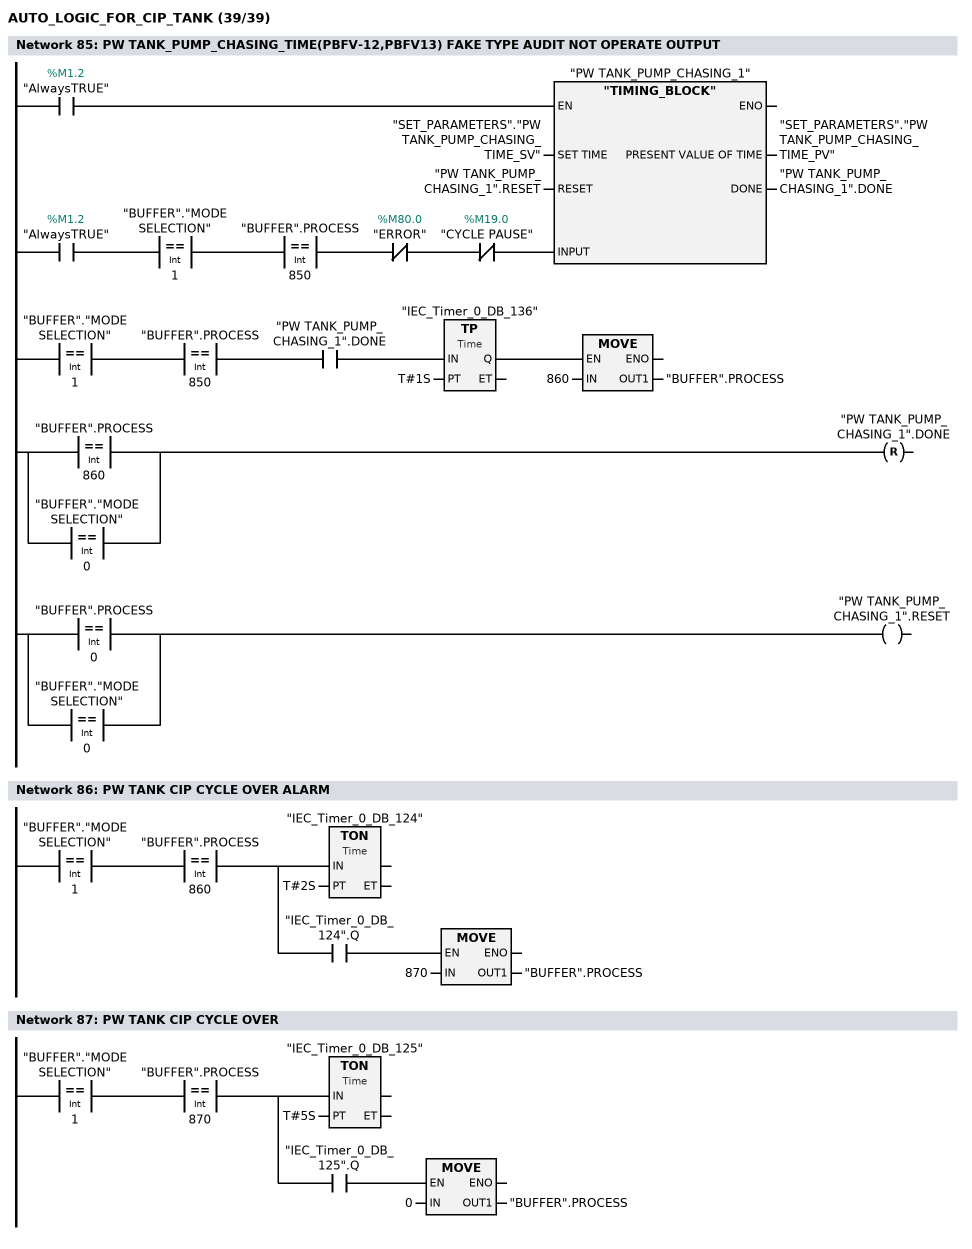
   RUNG wire#powerrail
      Contact( "AlwaysTRUE" )
      "PW TANK_PUMP_CHASING_1"(INPUT := wire#w1, "SET TIME" := "SET_PARAMETERS"."PW TANK_PUMP_CHASING_TIME_SV", RESET := "PW TANK_PUMP_CHASING_1".RESET, "PRESENT VALUE OF TIME" => "SET_PARAMETERS"."PW TANK_PUMP_CHASING_TIME_PV", DONE => "PW TANK_PUMP_CHASING_1".DONE)
   END_RUNG
   RUNG wire#powerrail
      Contact( "AlwaysTRUE" )
      { S7_Templates := "SrcType := Int" } EQ_Contact(in1 := "BUFFER"."MODE SELECTION", in2 := 1)
      { S7_Templates := "SrcType := Int" } EQ_Contact(in1 := "BUFFER".PROCESS, in2 := 850)
      I_Contact( "ERROR" )
      I_Contact( "CYCLE PAUSE" )
   END_RUNG wire#w1
   RUNG wire#powerrail
      { S7_Templates := "SrcType := Int" } EQ_Contact(in1 := "BUFFER"."MODE SELECTION", in2 := 1)
      { S7_Templates := "SrcType := Int" } EQ_Contact(in1 := "BUFFER".PROCESS, in2 := 850)
      Contact( "PW TANK_PUMP_CHASING_1".DONE )
      { S7_Templates := "time_type := Time" } "IEC_Timer_0_DB_136".TP(pt := T#1S, et =>)
      Move(in := 860, out1 => "BUFFER".PROCESS)
   END_RUNG
   RUNG wire#powerrail
      { S7_Templates := "SrcType := Int" } EQ_Contact(in1 := "BUFFER".PROCESS, in2 := 860)
      wire#w2
      R_Coil( "PW TANK_PUMP_CHASING_1".DONE )
   END_RUNG
   RUNG wire#powerrail
      { S7_Templates := "SrcType := Int" } EQ_Contact(in1 := "BUFFER"."MODE SELECTION", in2 := 0)
   END_RUNG wire#w2
   RUNG wire#powerrail
      { S7_Templates := "SrcType := Int" } EQ_Contact(in1 := "BUFFER".PROCESS, in2 := 0)
      wire#w3
      Coil( "PW TANK_PUMP_CHASING_1".RESET )
   END_RUNG
   RUNG wire#powerrail
      { S7_Templates := "SrcType := Int" } EQ_Contact(in1 := "BUFFER"."MODE SELECTION", in2 := 0)
   END_RUNG wire#w3
   // the same network as SCL:
   IF "AlwaysTRUE" THEN
       "PW TANK_PUMP_CHASING_1"("SET TIME" := "SET_PARAMETERS"."PW TANK_PUMP_CHASING_TIME_SV",   // "TIMING_BLOCK"
                               RESET := "PW TANK_PUMP_CHASING_1".RESET,
                               INPUT := "AlwaysTRUE" AND ("BUFFER"."MODE SELECTION" = 1) AND ("BUFFER".PROCESS = 850) AND NOT "ERROR" AND NOT "CYCLE PAUSE",
                               "PRESENT VALUE OF TIME" => "SET_PARAMETERS"."PW TANK_PUMP_CHASING_TIME_PV",
                               DONE => "PW TANK_PUMP_CHASING_1".DONE);
   END_IF;
   "IEC_Timer_0_DB_136".TP(IN := ("BUFFER"."MODE SELECTION" = 1) AND ("BUFFER".PROCESS = 850) AND "PW TANK_PUMP_CHASING_1".DONE,
                           PT := T#1S);
   IF "IEC_Timer_0_DB_136".Q THEN "BUFFER".PROCESS := 860; END_IF;
   IF ("BUFFER".PROCESS = 860) OR ("BUFFER"."MODE SELECTION" = 0) THEN
       "PW TANK_PUMP_CHASING_1".DONE := FALSE;
   END_IF;
   "PW TANK_PUMP_CHASING_1".RESET := ("BUFFER".PROCESS = 0) OR ("BUFFER"."MODE SELECTION" = 0);
END_REGION

REGION Network 86: PW TANK CIP CYCLE OVER ALARM
   RUNG wire#powerrail
      { S7_Templates := "SrcType := Int" } EQ_Contact(in1 := "BUFFER"."MODE SELECTION", in2 := 1)
      { S7_Templates := "SrcType := Int" } EQ_Contact(in1 := "BUFFER".PROCESS, in2 := 860)
      wire#w1
      { S7_Templates := "time_type := Time" } "IEC_Timer_0_DB_124".TON(pt := T#2S, et =>)
   END_RUNG
   RUNG wire#w1
      Contact( "IEC_Timer_0_DB_124".Q )
      Move(in := 870, out1 => "BUFFER".PROCESS)
   END_RUNG
   // the same network as SCL:
   #_w1 := ("BUFFER"."MODE SELECTION" = 1) AND ("BUFFER".PROCESS = 860);
   "IEC_Timer_0_DB_124".TON(IN := #_w1, PT := T#2S);
   IF #_w1 AND "IEC_Timer_0_DB_124".Q THEN "BUFFER".PROCESS := 870; END_IF;
END_REGION

REGION Network 87: PW TANK CIP CYCLE OVER
   RUNG wire#powerrail
      { S7_Templates := "SrcType := Int" } EQ_Contact(in1 := "BUFFER"."MODE SELECTION", in2 := 1)
      { S7_Templates := "SrcType := Int" } EQ_Contact(in1 := "BUFFER".PROCESS, in2 := 870)
      wire#w1
      { S7_Templates := "time_type := Time" } "IEC_Timer_0_DB_125".TON(pt := T#5S, et =>)
   END_RUNG
   RUNG wire#w1
      Contact( "IEC_Timer_0_DB_125".Q )
      Move(in := 0, out1 => "BUFFER".PROCESS)
   END_RUNG
   // the same network as SCL:
   #_w1 := ("BUFFER"."MODE SELECTION" = 1) AND ("BUFFER".PROCESS = 870);
   "IEC_Timer_0_DB_125".TON(IN := #_w1, PT := T#5S);
   IF #_w1 AND "IEC_Timer_0_DB_125".Q THEN "BUFFER".PROCESS := 0; END_IF;
END_REGION
END_FUNCTION

FUNCTION_BLOCK "TIMING_BLOCK"   // FB2, LAD
{ S7_Optimized_Access := 'TRUE' }
// stored: MemoryReserve 100, SetENOAutomatically false
   VAR_INPUT
      "SET TIME" : Int;
      RESET : Bool;
      INPUT : Bool;
   END_VAR
   VAR_OUTPUT
      "PRESENT VALUE OF TIME" : Int;
      DONE : Bool;
   END_VAR
   VAR
      "TIMER 1" { S7_SetPoint := 'True'} : IEC_TIMER;
   END_VAR
   VAR RETAIN
      "COUNTER1 1" { S7_SetPoint := 'True'} : IEC_COUNTER;
   END_VAR
   VAR_TEMP   // added for the SCL form of the ladder/FBD networks
      _w1 : Bool;
      _w2 : Bool;
   END_VAR
BEGIN

REGION Network 1
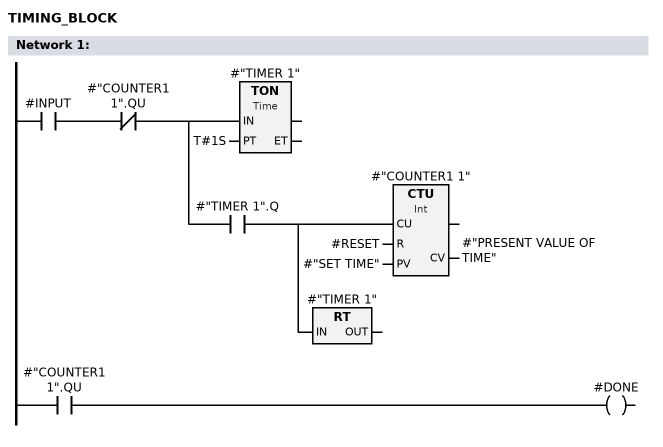
   RUNG wire#powerrail
      Contact( #INPUT )
      I_Contact( #"COUNTER1 1".QU )
      wire#w1
      { S7_Templates := "time_type := Time" } #"TIMER 1".TON(pt := T#1S, et =>)
   END_RUNG
   RUNG wire#w1
      Contact( #"TIMER 1".Q )
      wire#w2
      { S7_Templates := "value_type := Int" } #"COUNTER1 1".CTU(r := #RESET, pv := #"SET TIME", cv => #"PRESENT VALUE OF TIME")
   END_RUNG
   RUNG wire#w2
      RT_Coil( #"TIMER 1" )
   END_RUNG
   RUNG wire#powerrail
      Contact( #"COUNTER1 1".QU )
      Coil( #DONE )
   END_RUNG
   // the same network as SCL:
   #_w1 := #INPUT AND NOT #"COUNTER1 1".QU;
   #"TIMER 1".TON(IN := #_w1, PT := T#1S);
   #_w2 := #_w1 AND #"TIMER 1".Q;
   #"COUNTER1 1".CTU(CU := #_w2, R := #RESET, PV := #"SET TIME", CV => #"PRESENT VALUE OF TIME");
   IF #_w2 THEN RESET_TIMER(#"TIMER 1"); END_IF;
   #DONE := #"COUNTER1 1".QU;
END_REGION
END_FUNCTION_BLOCK

FUNCTION "POPUP" : Void   // FC6, LAD
{ S7_Optimized_Access := 'TRUE' }
// stored: SetENOAutomatically false
   VAR_TEMP   // added for the SCL form of the ladder/FBD networks
      _w1 : Bool;
      _w2 : Bool;
   END_VAR
BEGIN

REGION Network 1: RINSE-1_START
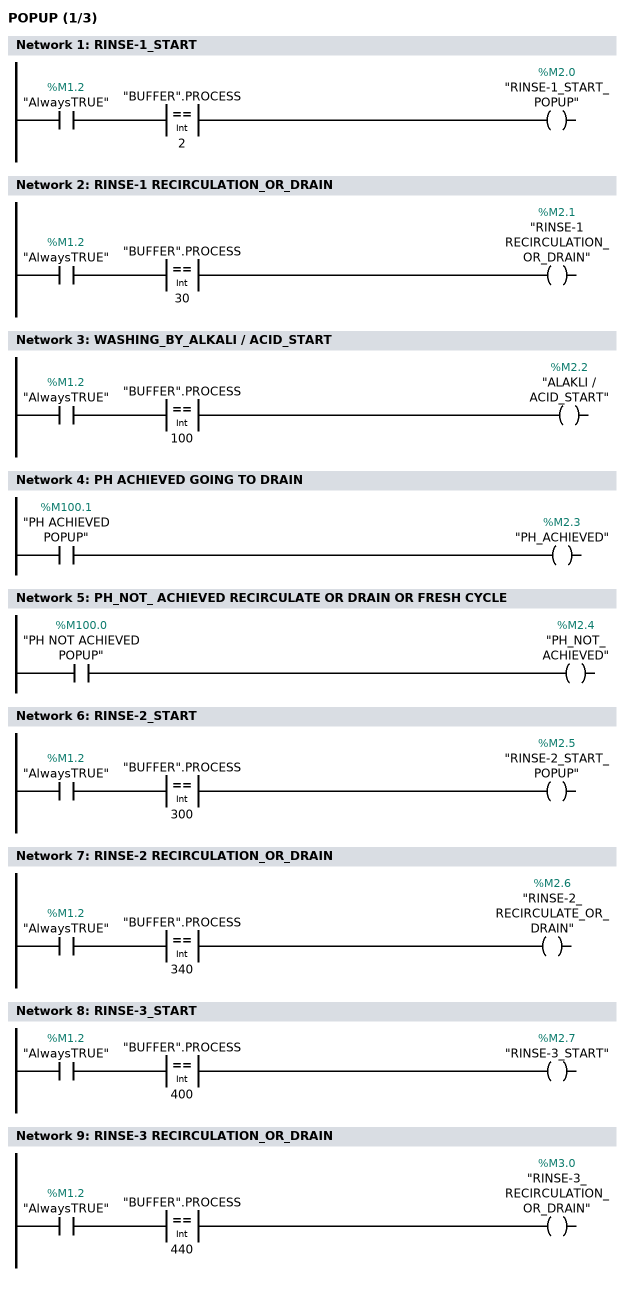
   RUNG wire#powerrail
      Contact( "AlwaysTRUE" )
      { S7_Templates := "SrcType := Int" } EQ_Contact(in1 := "BUFFER".PROCESS, in2 := 2)
      Coil( "RINSE-1_START_POPUP" )
   END_RUNG
   // the same network as SCL:
   "RINSE-1_START_POPUP" := "AlwaysTRUE" AND ("BUFFER".PROCESS = 2);
END_REGION

REGION Network 2: RINSE-1 RECIRCULATION_OR_DRAIN
   RUNG wire#powerrail
      Contact( "AlwaysTRUE" )
      { S7_Templates := "SrcType := Int" } EQ_Contact(in1 := "BUFFER".PROCESS, in2 := 30)
      Coil( "RINSE-1 RECIRCULATION_OR_DRAIN" )
   END_RUNG
   // the same network as SCL:
   "RINSE-1 RECIRCULATION_OR_DRAIN" := "AlwaysTRUE" AND ("BUFFER".PROCESS = 30);
END_REGION

REGION Network 3: WASHING_BY_ALKALI / ACID_START
   RUNG wire#powerrail
      Contact( "AlwaysTRUE" )
      { S7_Templates := "SrcType := Int" } EQ_Contact(in1 := "BUFFER".PROCESS, in2 := 100)
      Coil( "ALAKLI / ACID_START" )
   END_RUNG
   // the same network as SCL:
   "ALAKLI / ACID_START" := "AlwaysTRUE" AND ("BUFFER".PROCESS = 100);
END_REGION

REGION Network 4: PH ACHIEVED GOING TO DRAIN
   RUNG wire#powerrail
      Contact( "PH ACHIEVED POPUP" )
      Coil( "PH_ACHIEVED" )
   END_RUNG
   // the same network as SCL:
   "PH_ACHIEVED" := "PH ACHIEVED POPUP";
END_REGION

REGION Network 5: PH_NOT_ ACHIEVED RECIRCULATE OR DRAIN OR FRESH CYCLE
   RUNG wire#powerrail
      Contact( "PH NOT ACHIEVED POPUP" )
      Coil( "PH_NOT_ACHIEVED" )
   END_RUNG
   // the same network as SCL:
   "PH_NOT_ACHIEVED" := "PH NOT ACHIEVED POPUP";
END_REGION

REGION Network 6: RINSE-2_START
   RUNG wire#powerrail
      Contact( "AlwaysTRUE" )
      { S7_Templates := "SrcType := Int" } EQ_Contact(in1 := "BUFFER".PROCESS, in2 := 300)
      Coil( "RINSE-2_START_POPUP" )
   END_RUNG
   // the same network as SCL:
   "RINSE-2_START_POPUP" := "AlwaysTRUE" AND ("BUFFER".PROCESS = 300);
END_REGION

REGION Network 7: RINSE-2 RECIRCULATION_OR_DRAIN
   RUNG wire#powerrail
      Contact( "AlwaysTRUE" )
      { S7_Templates := "SrcType := Int" } EQ_Contact(in1 := "BUFFER".PROCESS, in2 := 340)
      Coil( "RINSE-2_RECIRCULATE_OR_DRAIN" )
   END_RUNG
   // the same network as SCL:
   "RINSE-2_RECIRCULATE_OR_DRAIN" := "AlwaysTRUE" AND ("BUFFER".PROCESS = 340);
END_REGION

REGION Network 8: RINSE-3_START
   RUNG wire#powerrail
      Contact( "AlwaysTRUE" )
      { S7_Templates := "SrcType := Int" } EQ_Contact(in1 := "BUFFER".PROCESS, in2 := 400)
      Coil( "RINSE-3_START" )
   END_RUNG
   // the same network as SCL:
   "RINSE-3_START" := "AlwaysTRUE" AND ("BUFFER".PROCESS = 400);
END_REGION

REGION Network 9: RINSE-3 RECIRCULATION_OR_DRAIN
   RUNG wire#powerrail
      Contact( "AlwaysTRUE" )
      { S7_Templates := "SrcType := Int" } EQ_Contact(in1 := "BUFFER".PROCESS, in2 := 440)
      Coil( "RINSE-3_RECIRCULATION_OR_DRAIN" )
   END_RUNG
   // the same network as SCL:
   "RINSE-3_RECIRCULATION_OR_DRAIN" := "AlwaysTRUE" AND ("BUFFER".PROCESS = 440);
END_REGION

REGION Network 10: FINAL_RINSE_START
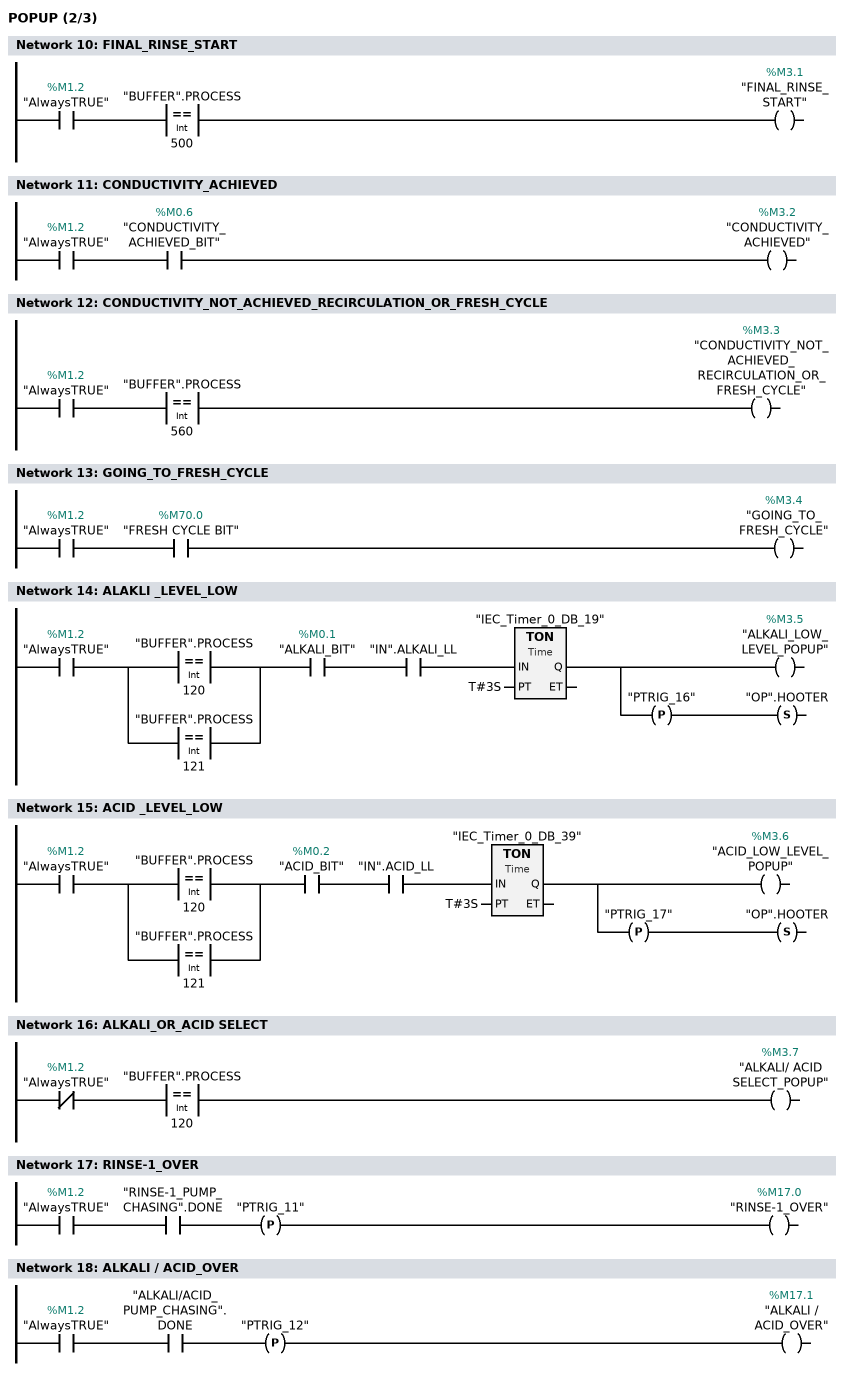
   RUNG wire#powerrail
      Contact( "AlwaysTRUE" )
      { S7_Templates := "SrcType := Int" } EQ_Contact(in1 := "BUFFER".PROCESS, in2 := 500)
      Coil( "FINAL_RINSE_START" )
   END_RUNG
   // the same network as SCL:
   "FINAL_RINSE_START" := "AlwaysTRUE" AND ("BUFFER".PROCESS = 500);
END_REGION

REGION Network 11: CONDUCTIVITY_ACHIEVED
   RUNG wire#powerrail
      Contact( "AlwaysTRUE" )
      Contact( "CONDUCTIVITY_ACHIEVED_BIT" )
      Coil( "CONDUCTIVITY_ACHIEVED" )
   END_RUNG
   // the same network as SCL:
   "CONDUCTIVITY_ACHIEVED" := "AlwaysTRUE" AND "CONDUCTIVITY_ACHIEVED_BIT";
END_REGION

REGION Network 12: CONDUCTIVITY_NOT_ACHIEVED_RECIRCULATION_OR_FRESH_CYCLE
   RUNG wire#powerrail
      Contact( "AlwaysTRUE" )
      { S7_Templates := "SrcType := Int" } EQ_Contact(in1 := "BUFFER".PROCESS, in2 := 560)
      Coil( "CONDUCTIVITY_NOT_ACHIEVED_RECIRCULATION_OR_FRESH_CYCLE" )
   END_RUNG
   // the same network as SCL:
   "CONDUCTIVITY_NOT_ACHIEVED_RECIRCULATION_OR_FRESH_CYCLE" := "AlwaysTRUE" AND ("BUFFER".PROCESS = 560);
END_REGION

REGION Network 13: GOING_TO_FRESH_CYCLE
   RUNG wire#powerrail
      Contact( "AlwaysTRUE" )
      Contact( "FRESH CYCLE BIT" )
      Coil( "GOING_TO_FRESH_CYCLE" )
   END_RUNG
   // the same network as SCL:
   "GOING_TO_FRESH_CYCLE" := "AlwaysTRUE" AND "FRESH CYCLE BIT";
END_REGION

REGION Network 14: ALAKLI _LEVEL_LOW
   RUNG wire#powerrail
      Contact( "AlwaysTRUE" )
      wire#w1
      { S7_Templates := "SrcType := Int" } EQ_Contact(in1 := "BUFFER".PROCESS, in2 := 120)
      wire#w2
      Contact( "ALKALI_BIT" )
      Contact( "IN".ALKALI_LL )
      { S7_Templates := "time_type := Time" } "IEC_Timer_0_DB_19".TON(pt := T#3S, et =>)
      wire#w3
      Coil( "ALKALI_LOW_LEVEL_POPUP" )
   END_RUNG
   RUNG wire#w1
      { S7_Templates := "SrcType := Int" } EQ_Contact(in1 := "BUFFER".PROCESS, in2 := 121)
   END_RUNG wire#w2
   RUNG wire#w3
      P_Trig( "PTRIG_16" )
      S_Coil( "OP".HOOTER )
   END_RUNG
   // the same network as SCL:
   "IEC_Timer_0_DB_19".TON(IN := "AlwaysTRUE" AND (("BUFFER".PROCESS = 120) OR ("BUFFER".PROCESS = 121)) AND "ALKALI_BIT" AND "IN".ALKALI_LL,
                           PT := T#3S);
   "ALKALI_LOW_LEVEL_POPUP" := "IEC_Timer_0_DB_19".Q;
   #_w1 := "IEC_Timer_0_DB_19".Q AND NOT "PTRIG_16";   // rising edge
   "PTRIG_16" := "IEC_Timer_0_DB_19".Q;
   IF #_w1 THEN "OP".HOOTER := TRUE; END_IF;
END_REGION

REGION Network 15: ACID _LEVEL_LOW
   RUNG wire#powerrail
      Contact( "AlwaysTRUE" )
      wire#w1
      { S7_Templates := "SrcType := Int" } EQ_Contact(in1 := "BUFFER".PROCESS, in2 := 120)
      wire#w2
      Contact( "ACID_BIT" )
      Contact( "IN".ACID_LL )
      { S7_Templates := "time_type := Time" } "IEC_Timer_0_DB_39".TON(pt := T#3S, et =>)
      wire#w3
      Coil( "ACID_LOW_LEVEL_POPUP" )
   END_RUNG
   RUNG wire#w1
      { S7_Templates := "SrcType := Int" } EQ_Contact(in1 := "BUFFER".PROCESS, in2 := 121)
   END_RUNG wire#w2
   RUNG wire#w3
      P_Trig( "PTRIG_17" )
      S_Coil( "OP".HOOTER )
   END_RUNG
   // the same network as SCL:
   "IEC_Timer_0_DB_39".TON(IN := "AlwaysTRUE" AND (("BUFFER".PROCESS = 120) OR ("BUFFER".PROCESS = 121)) AND "ACID_BIT" AND "IN".ACID_LL,
                           PT := T#3S);
   "ACID_LOW_LEVEL_POPUP" := "IEC_Timer_0_DB_39".Q;
   #_w1 := "IEC_Timer_0_DB_39".Q AND NOT "PTRIG_17";   // rising edge
   "PTRIG_17" := "IEC_Timer_0_DB_39".Q;
   IF #_w1 THEN "OP".HOOTER := TRUE; END_IF;
END_REGION

REGION Network 16: ALKALI_OR_ACID SELECT
   RUNG wire#powerrail
      I_Contact( "AlwaysTRUE" )
      { S7_Templates := "SrcType := Int" } EQ_Contact(in1 := "BUFFER".PROCESS, in2 := 120)
      Coil( "ALKALI/ ACID SELECT_POPUP" )
   END_RUNG
   // the same network as SCL:
   "ALKALI/ ACID SELECT_POPUP" := NOT "AlwaysTRUE" AND ("BUFFER".PROCESS = 120);
END_REGION

REGION Network 17: RINSE-1_OVER
   RUNG wire#powerrail
      Contact( "AlwaysTRUE" )
      Contact( "RINSE-1_PUMP_CHASING".DONE )
      P_Trig( "PTRIG_11" )
      Coil( "RINSE-1_OVER" )
   END_RUNG
   // the same network as SCL:
   #_w1 := "AlwaysTRUE" AND "RINSE-1_PUMP_CHASING".DONE;
   #_w2 := #_w1 AND NOT "PTRIG_11";   // rising edge
   "PTRIG_11" := #_w1;
   "RINSE-1_OVER" := #_w2;
END_REGION

REGION Network 18: ALKALI / ACID_OVER
   RUNG wire#powerrail
      Contact( "AlwaysTRUE" )
      Contact( "ALKALI/ACID_PUMP_CHASING".DONE )
      P_Trig( "PTRIG_12" )
      Coil( "ALKALI / ACID_OVER" )
   END_RUNG
   // the same network as SCL:
   #_w1 := "AlwaysTRUE" AND "ALKALI/ACID_PUMP_CHASING".DONE;
   #_w2 := #_w1 AND NOT "PTRIG_12";   // rising edge
   "PTRIG_12" := #_w1;
   "ALKALI / ACID_OVER" := #_w2;
END_REGION

REGION Network 19: RINSE-2_OVER
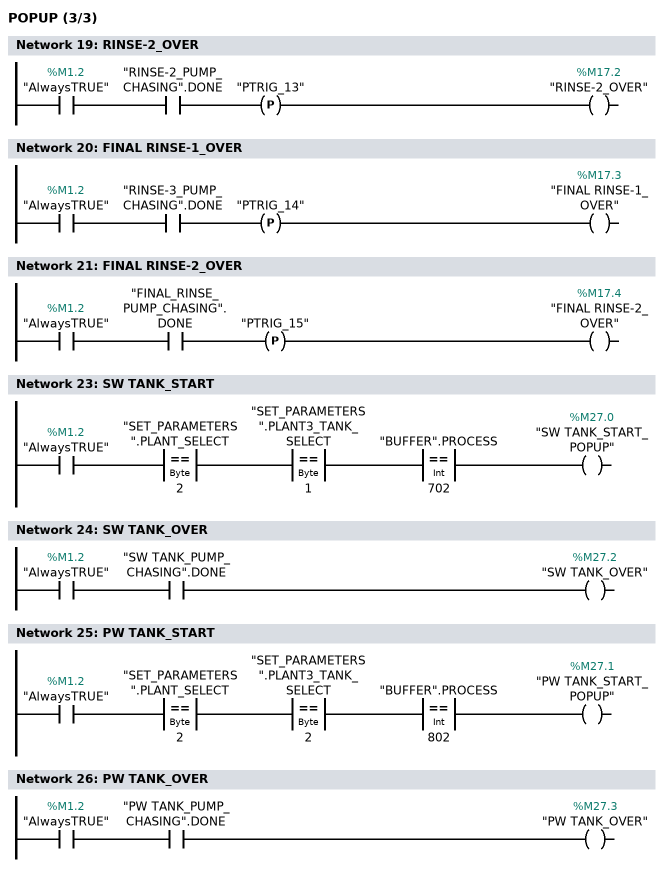
   RUNG wire#powerrail
      Contact( "AlwaysTRUE" )
      Contact( "RINSE-2_PUMP_CHASING".DONE )
      P_Trig( "PTRIG_13" )
      Coil( "RINSE-2_OVER" )
   END_RUNG
   // the same network as SCL:
   #_w1 := "AlwaysTRUE" AND "RINSE-2_PUMP_CHASING".DONE;
   #_w2 := #_w1 AND NOT "PTRIG_13";   // rising edge
   "PTRIG_13" := #_w1;
   "RINSE-2_OVER" := #_w2;
END_REGION

REGION Network 20: FINAL RINSE-1_OVER
   RUNG wire#powerrail
      Contact( "AlwaysTRUE" )
      Contact( "RINSE-3_PUMP_CHASING".DONE )
      P_Trig( "PTRIG_14" )
      Coil( "FINAL RINSE-1_OVER" )
   END_RUNG
   // the same network as SCL:
   #_w1 := "AlwaysTRUE" AND "RINSE-3_PUMP_CHASING".DONE;
   #_w2 := #_w1 AND NOT "PTRIG_14";   // rising edge
   "PTRIG_14" := #_w1;
   "FINAL RINSE-1_OVER" := #_w2;
END_REGION

REGION Network 21: FINAL RINSE-2_OVER
   RUNG wire#powerrail
      Contact( "AlwaysTRUE" )
      Contact( "FINAL_RINSE_PUMP_CHASING".DONE )
      P_Trig( "PTRIG_15" )
      Coil( "FINAL RINSE-2_OVER" )
   END_RUNG
   // the same network as SCL:
   #_w1 := "AlwaysTRUE" AND "FINAL_RINSE_PUMP_CHASING".DONE;
   #_w2 := #_w1 AND NOT "PTRIG_15";   // rising edge
   "PTRIG_15" := #_w1;
   "FINAL RINSE-2_OVER" := #_w2;
END_REGION

REGION Network 22: ------------NEW LOGIC ADD-----------
END_REGION

REGION Network 23: SW TANK_START
   RUNG wire#powerrail
      Contact( "AlwaysTRUE" )
      { S7_Templates := "SrcType := Byte" } EQ_Contact(in1 := "SET_PARAMETERS".PLANT_SELECT, in2 := 2)
      { S7_Templates := "SrcType := Byte" } EQ_Contact(in1 := "SET_PARAMETERS".PLANT3_TANK_SELECT, in2 := 1)
      { S7_Templates := "SrcType := Int" } EQ_Contact(in1 := "BUFFER".PROCESS, in2 := 702)
      Coil( "SW TANK_START_POPUP" )
   END_RUNG
   // the same network as SCL:
   "SW TANK_START_POPUP" := "AlwaysTRUE" AND ("SET_PARAMETERS".PLANT_SELECT = 2) AND ("SET_PARAMETERS".PLANT3_TANK_SELECT = 1) AND ("BUFFER".PROCESS = 702);
END_REGION

REGION Network 24: SW TANK_OVER
   RUNG wire#powerrail
      Contact( "AlwaysTRUE" )
      Contact( "SW TANK_PUMP_CHASING".DONE )
      Coil( "SW TANK_OVER" )
   END_RUNG
   // the same network as SCL:
   "SW TANK_OVER" := "AlwaysTRUE" AND "SW TANK_PUMP_CHASING".DONE;
END_REGION

REGION Network 25: PW TANK_START
   RUNG wire#powerrail
      Contact( "AlwaysTRUE" )
      { S7_Templates := "SrcType := Byte" } EQ_Contact(in1 := "SET_PARAMETERS".PLANT_SELECT, in2 := 2)
      { S7_Templates := "SrcType := Byte" } EQ_Contact(in1 := "SET_PARAMETERS".PLANT3_TANK_SELECT, in2 := 2)
      { S7_Templates := "SrcType := Int" } EQ_Contact(in1 := "BUFFER".PROCESS, in2 := 802)
      Coil( "PW TANK_START_POPUP" )
   END_RUNG
   // the same network as SCL:
   "PW TANK_START_POPUP" := "AlwaysTRUE" AND ("SET_PARAMETERS".PLANT_SELECT = 2) AND ("SET_PARAMETERS".PLANT3_TANK_SELECT = 2) AND ("BUFFER".PROCESS = 802);
END_REGION

REGION Network 26: PW TANK_OVER
   RUNG wire#powerrail
      Contact( "AlwaysTRUE" )
      Contact( "PW TANK_PUMP_CHASING".DONE )
      Coil( "PW TANK_OVER" )
   END_RUNG
   // the same network as SCL:
   "PW TANK_OVER" := "AlwaysTRUE" AND "PW TANK_PUMP_CHASING".DONE;
END_REGION
END_FUNCTION

FUNCTION "SCALING_PARAMETERS" : Void   // FC4, LAD
{ S7_Optimized_Access := 'TRUE' }
// stored: SetENOAutomatically false
BEGIN

REGION Network 1: PH_SCALE
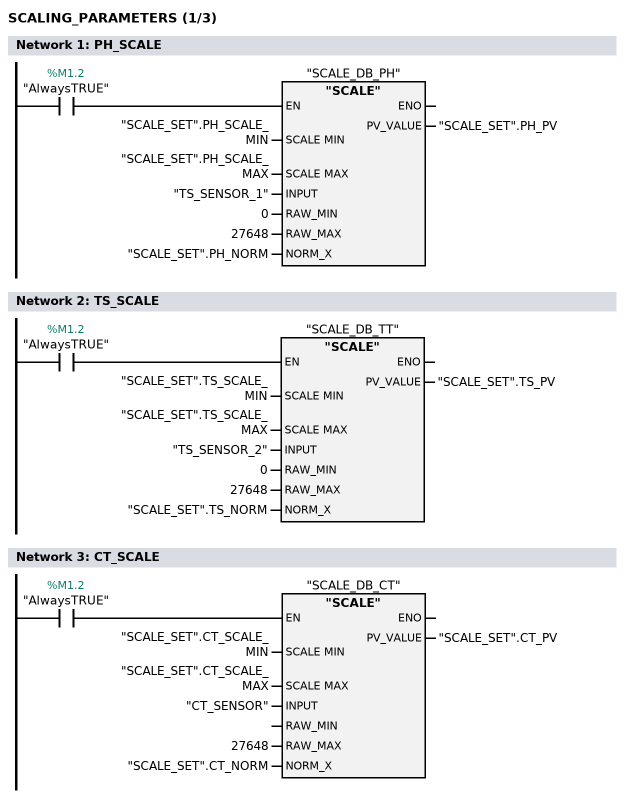
   RUNG wire#powerrail
      Contact( "AlwaysTRUE" )
      "SCALE_DB_PH"("SCALE MIN" := "SCALE_SET".PH_SCALE_MIN, "SCALE MAX" := "SCALE_SET".PH_SCALE_MAX, INPUT := "TS_SENSOR_1", RAW_MIN := 0, RAW_MAX := 27648, NORM_X := "SCALE_SET".PH_NORM, PV_VALUE => "SCALE_SET".PH_PV)
   END_RUNG
   // the same network as SCL:
   IF "AlwaysTRUE" THEN
       "SCALE_DB_PH"("SCALE MIN" := "SCALE_SET".PH_SCALE_MIN,   // "SCALE"
                     "SCALE MAX" := "SCALE_SET".PH_SCALE_MAX,
                     INPUT := "TS_SENSOR_1",
                     RAW_MIN := 0,
                     RAW_MAX := 27648,
                     NORM_X := "SCALE_SET".PH_NORM,
                     PV_VALUE => "SCALE_SET".PH_PV);
   END_IF;
END_REGION

REGION Network 2: TS_SCALE
   RUNG wire#powerrail
      Contact( "AlwaysTRUE" )
      "SCALE_DB_TT"("SCALE MIN" := "SCALE_SET".TS_SCALE_MIN, "SCALE MAX" := "SCALE_SET".TS_SCALE_MAX, INPUT := "TS_SENSOR_2", RAW_MIN := 0, RAW_MAX := 27648, NORM_X := "SCALE_SET".TS_NORM, PV_VALUE => "SCALE_SET".TS_PV)
   END_RUNG
   // the same network as SCL:
   IF "AlwaysTRUE" THEN
       "SCALE_DB_TT"("SCALE MIN" := "SCALE_SET".TS_SCALE_MIN,   // "SCALE"
                     "SCALE MAX" := "SCALE_SET".TS_SCALE_MAX,
                     INPUT := "TS_SENSOR_2",
                     RAW_MIN := 0,
                     RAW_MAX := 27648,
                     NORM_X := "SCALE_SET".TS_NORM,
                     PV_VALUE => "SCALE_SET".TS_PV);
   END_IF;
END_REGION

REGION Network 3: CT_SCALE
   RUNG wire#powerrail
      Contact( "AlwaysTRUE" )
      "SCALE_DB_CT"("SCALE MIN" := "SCALE_SET".CT_SCALE_MIN, "SCALE MAX" := "SCALE_SET".CT_SCALE_MAX, INPUT := "CT_SENSOR", RAW_MIN :=, RAW_MAX := 27648, NORM_X := "SCALE_SET".CT_NORM, PV_VALUE => "SCALE_SET".CT_PV)
   END_RUNG
   // the same network as SCL:
   IF "AlwaysTRUE" THEN
       "SCALE_DB_CT"("SCALE MIN" := "SCALE_SET".CT_SCALE_MIN,   // "SCALE"
                     "SCALE MAX" := "SCALE_SET".CT_SCALE_MAX,
                     INPUT := "CT_SENSOR",
                     RAW_MAX := 27648,
                     NORM_X := "SCALE_SET".CT_NORM,
                     PV_VALUE => "SCALE_SET".CT_PV);
   END_IF;
END_REGION

REGION Network 4: SET_PUMP_SPEED
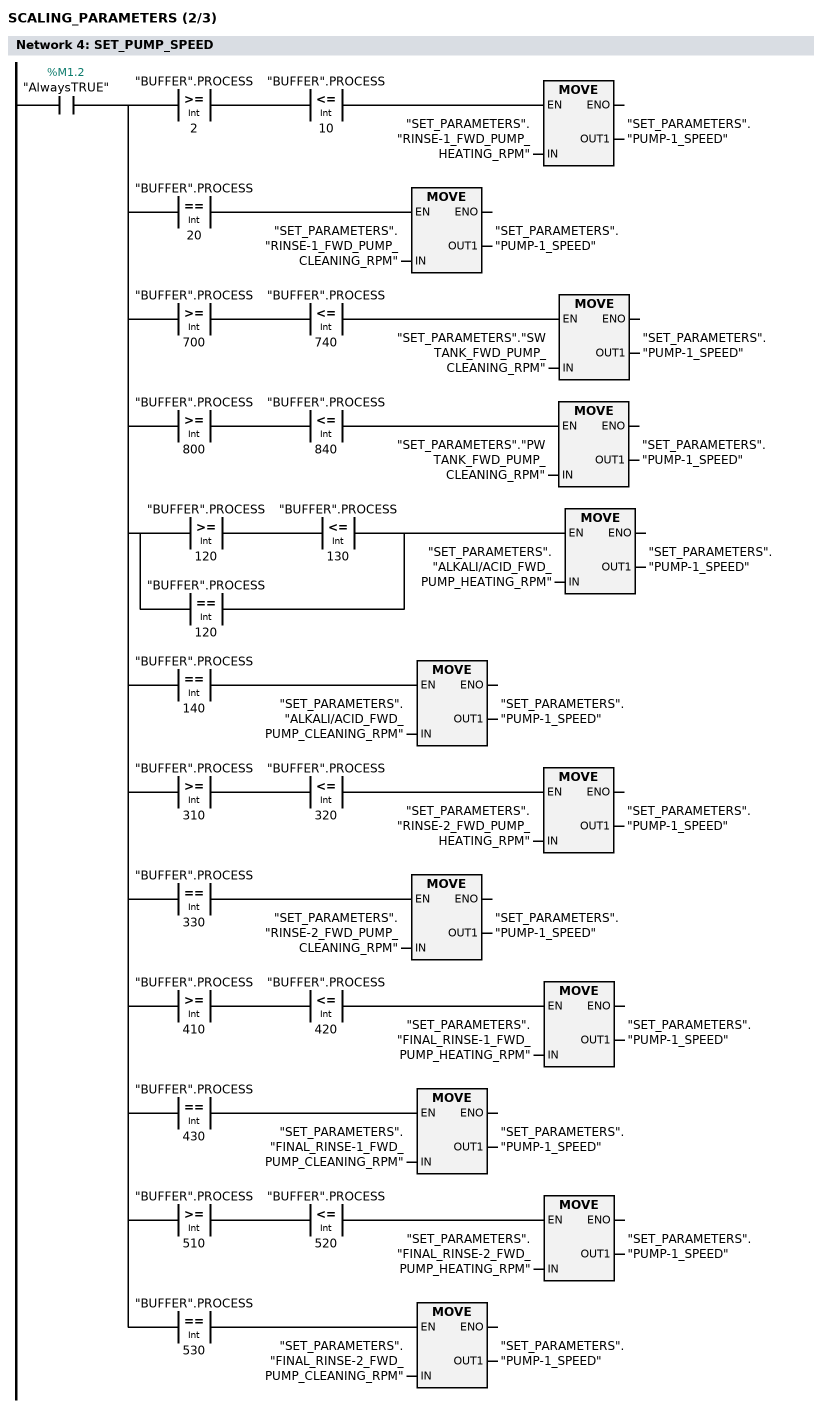
   RUNG wire#powerrail
      Contact( "AlwaysTRUE" )
      wire#w1
      { S7_Templates := "SrcType := Int" } GE_Contact(in1 := "BUFFER".PROCESS, in2 := 2)
      { S7_Templates := "SrcType := Int" } LE_Contact(in1 := "BUFFER".PROCESS, in2 := 10)
      Move(in := "SET_PARAMETERS"."RINSE-1_FWD_PUMP_HEATING_RPM", out1 => "SET_PARAMETERS"."PUMP-1_SPEED")
   END_RUNG
   RUNG wire#w1
      { S7_Templates := "SrcType := Int" } EQ_Contact(in1 := "BUFFER".PROCESS, in2 := 20)
      Move(in := "SET_PARAMETERS"."RINSE-1_FWD_PUMP_CLEANING_RPM", out1 => "SET_PARAMETERS"."PUMP-1_SPEED")
   END_RUNG
   RUNG wire#w1
      { S7_Templates := "SrcType := Int" } GE_Contact(in1 := "BUFFER".PROCESS, in2 := 700)
      { S7_Templates := "SrcType := Int" } LE_Contact(in1 := "BUFFER".PROCESS, in2 := 740)
      Move(in := "SET_PARAMETERS"."SW TANK_FWD_PUMP_CLEANING_RPM", out1 => "SET_PARAMETERS"."PUMP-1_SPEED")
   END_RUNG
   RUNG wire#w1
      { S7_Templates := "SrcType := Int" } GE_Contact(in1 := "BUFFER".PROCESS, in2 := 800)
      { S7_Templates := "SrcType := Int" } LE_Contact(in1 := "BUFFER".PROCESS, in2 := 840)
      Move(in := "SET_PARAMETERS"."PW TANK_FWD_PUMP_CLEANING_RPM", out1 => "SET_PARAMETERS"."PUMP-1_SPEED")
   END_RUNG
   RUNG wire#w1
      { S7_Templates := "SrcType := Int" } GE_Contact(in1 := "BUFFER".PROCESS, in2 := 120)
      { S7_Templates := "SrcType := Int" } LE_Contact(in1 := "BUFFER".PROCESS, in2 := 130)
      wire#w2
      Move(in := "SET_PARAMETERS"."ALKALI/ACID_FWD_PUMP_HEATING_RPM", out1 => "SET_PARAMETERS"."PUMP-1_SPEED")
   END_RUNG
   RUNG wire#w1
      { S7_Templates := "SrcType := Int" } EQ_Contact(in1 := "BUFFER".PROCESS, in2 := 120)
   END_RUNG wire#w2
   RUNG wire#w1
      { S7_Templates := "SrcType := Int" } EQ_Contact(in1 := "BUFFER".PROCESS, in2 := 140)
      Move(in := "SET_PARAMETERS"."ALKALI/ACID_FWD_PUMP_CLEANING_RPM", out1 => "SET_PARAMETERS"."PUMP-1_SPEED")
   END_RUNG
   RUNG wire#w1
      { S7_Templates := "SrcType := Int" } GE_Contact(in1 := "BUFFER".PROCESS, in2 := 310)
      { S7_Templates := "SrcType := Int" } LE_Contact(in1 := "BUFFER".PROCESS, in2 := 320)
      Move(in := "SET_PARAMETERS"."RINSE-2_FWD_PUMP_HEATING_RPM", out1 => "SET_PARAMETERS"."PUMP-1_SPEED")
   END_RUNG
   RUNG wire#w1
      { S7_Templates := "SrcType := Int" } EQ_Contact(in1 := "BUFFER".PROCESS, in2 := 330)
      Move(in := "SET_PARAMETERS"."RINSE-2_FWD_PUMP_CLEANING_RPM", out1 => "SET_PARAMETERS"."PUMP-1_SPEED")
   END_RUNG
   RUNG wire#w1
      { S7_Templates := "SrcType := Int" } GE_Contact(in1 := "BUFFER".PROCESS, in2 := 410)
      { S7_Templates := "SrcType := Int" } LE_Contact(in1 := "BUFFER".PROCESS, in2 := 420)
      Move(in := "SET_PARAMETERS"."FINAL_RINSE-1_FWD_PUMP_HEATING_RPM", out1 => "SET_PARAMETERS"."PUMP-1_SPEED")
   END_RUNG
   RUNG wire#w1
      { S7_Templates := "SrcType := Int" } EQ_Contact(in1 := "BUFFER".PROCESS, in2 := 430)
      Move(in := "SET_PARAMETERS"."FINAL_RINSE-1_FWD_PUMP_CLEANING_RPM", out1 => "SET_PARAMETERS"."PUMP-1_SPEED")
   END_RUNG
   RUNG wire#w1
      { S7_Templates := "SrcType := Int" } GE_Contact(in1 := "BUFFER".PROCESS, in2 := 510)
      { S7_Templates := "SrcType := Int" } LE_Contact(in1 := "BUFFER".PROCESS, in2 := 520)
      Move(in := "SET_PARAMETERS"."FINAL_RINSE-2_FWD_PUMP_HEATING_RPM", out1 => "SET_PARAMETERS"."PUMP-1_SPEED")
   END_RUNG
   RUNG wire#w1
      { S7_Templates := "SrcType := Int" } EQ_Contact(in1 := "BUFFER".PROCESS, in2 := 530)
      Move(in := "SET_PARAMETERS"."FINAL_RINSE-2_FWD_PUMP_CLEANING_RPM", out1 => "SET_PARAMETERS"."PUMP-1_SPEED")
   END_RUNG
   // the same network as SCL:
   IF "AlwaysTRUE" AND ("BUFFER".PROCESS >= 2) AND ("BUFFER".PROCESS <= 10) THEN
       "SET_PARAMETERS"."PUMP-1_SPEED" := "SET_PARAMETERS"."RINSE-1_FWD_PUMP_HEATING_RPM";
   END_IF;
   IF "AlwaysTRUE" AND ("BUFFER".PROCESS = 20) THEN
       "SET_PARAMETERS"."PUMP-1_SPEED" := "SET_PARAMETERS"."RINSE-1_FWD_PUMP_CLEANING_RPM";
   END_IF;
   IF "AlwaysTRUE" AND ("BUFFER".PROCESS >= 700) AND ("BUFFER".PROCESS <= 740) THEN
       "SET_PARAMETERS"."PUMP-1_SPEED" := "SET_PARAMETERS"."SW TANK_FWD_PUMP_CLEANING_RPM";
   END_IF;
   IF "AlwaysTRUE" AND ("BUFFER".PROCESS >= 800) AND ("BUFFER".PROCESS <= 840) THEN
       "SET_PARAMETERS"."PUMP-1_SPEED" := "SET_PARAMETERS"."PW TANK_FWD_PUMP_CLEANING_RPM";
   END_IF;
   IF "AlwaysTRUE" AND ((("BUFFER".PROCESS >= 120) AND ("BUFFER".PROCESS <= 130)) OR ("BUFFER".PROCESS = 120)) THEN
       "SET_PARAMETERS"."PUMP-1_SPEED" := "SET_PARAMETERS"."ALKALI/ACID_FWD_PUMP_HEATING_RPM";
   END_IF;
   IF "AlwaysTRUE" AND ("BUFFER".PROCESS = 140) THEN
       "SET_PARAMETERS"."PUMP-1_SPEED" := "SET_PARAMETERS"."ALKALI/ACID_FWD_PUMP_CLEANING_RPM";
   END_IF;
   IF "AlwaysTRUE" AND ("BUFFER".PROCESS >= 310) AND ("BUFFER".PROCESS <= 320) THEN
       "SET_PARAMETERS"."PUMP-1_SPEED" := "SET_PARAMETERS"."RINSE-2_FWD_PUMP_HEATING_RPM";
   END_IF;
   IF "AlwaysTRUE" AND ("BUFFER".PROCESS = 330) THEN
       "SET_PARAMETERS"."PUMP-1_SPEED" := "SET_PARAMETERS"."RINSE-2_FWD_PUMP_CLEANING_RPM";
   END_IF;
   IF "AlwaysTRUE" AND ("BUFFER".PROCESS >= 410) AND ("BUFFER".PROCESS <= 420) THEN
       "SET_PARAMETERS"."PUMP-1_SPEED" := "SET_PARAMETERS"."FINAL_RINSE-1_FWD_PUMP_HEATING_RPM";
   END_IF;
   IF "AlwaysTRUE" AND ("BUFFER".PROCESS = 430) THEN
       "SET_PARAMETERS"."PUMP-1_SPEED" := "SET_PARAMETERS"."FINAL_RINSE-1_FWD_PUMP_CLEANING_RPM";
   END_IF;
   IF "AlwaysTRUE" AND ("BUFFER".PROCESS >= 510) AND ("BUFFER".PROCESS <= 520) THEN
       "SET_PARAMETERS"."PUMP-1_SPEED" := "SET_PARAMETERS"."FINAL_RINSE-2_FWD_PUMP_HEATING_RPM";
   END_IF;
   IF "AlwaysTRUE" AND ("BUFFER".PROCESS = 530) THEN
       "SET_PARAMETERS"."PUMP-1_SPEED" := "SET_PARAMETERS"."FINAL_RINSE-2_FWD_PUMP_CLEANING_RPM";
   END_IF;
END_REGION

REGION Network 5: PUMP-1 SPEED
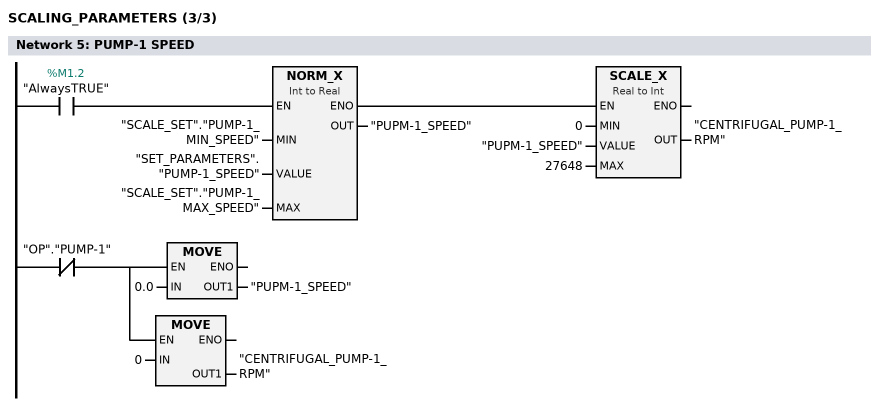
   RUNG wire#powerrail
      Contact( "AlwaysTRUE" )
      { S7_Templates := "[SrcType := Int, DestType := Real]" } Normalize(min := "SCALE_SET"."PUMP-1_MIN_SPEED", value := "SET_PARAMETERS"."PUMP-1_SPEED", max := "SCALE_SET"."PUMP-1_MAX_SPEED", out => "PUPM-1_SPEED")
      { S7_Templates := "[SrcType := Real, DestType := Int]" } Scale(min := 0, value := "PUPM-1_SPEED", max := 27648, out => "CENTRIFUGAL_PUMP-1_RPM")
   END_RUNG
   RUNG wire#powerrail
      I_Contact( "OP"."PUMP-1" )
      wire#w1
      Move(in := 0.0, out1 => "PUPM-1_SPEED")
   END_RUNG
   RUNG wire#w1
      Move(in := 0, out1 => "CENTRIFUGAL_PUMP-1_RPM")
   END_RUNG
   // the same network as SCL:
   IF "AlwaysTRUE" THEN
       "PUPM-1_SPEED" := NORM_X(MIN := "SCALE_SET"."PUMP-1_MIN_SPEED", VALUE := "SET_PARAMETERS"."PUMP-1_SPEED", MAX := "SCALE_SET"."PUMP-1_MAX_SPEED");
       "CENTRIFUGAL_PUMP-1_RPM" := SCALE_X(MIN := 0, VALUE := "PUPM-1_SPEED", MAX := 27648);
   END_IF;
   IF NOT "OP"."PUMP-1" THEN
       "PUPM-1_SPEED" := 0.0;
       "CENTRIFUGAL_PUMP-1_RPM" := 0;
   END_IF;
END_REGION
END_FUNCTION

FUNCTION_BLOCK "SCALE"   // FB1, LAD
{ S7_Optimized_Access := 'TRUE' }
// stored: MemoryReserve 100, SetENOAutomatically false
   VAR_INPUT
      "SCALE MIN" : Real;
      "SCALE MAX" : Real;
      INPUT : Int;
      RAW_MIN : Int;
      RAW_MAX : Int;
   END_VAR
   VAR_OUTPUT
      PV_VALUE : Real;
   END_VAR
   VAR_IN_OUT
      NORM_X : Real;
   END_VAR
BEGIN

REGION Network 1
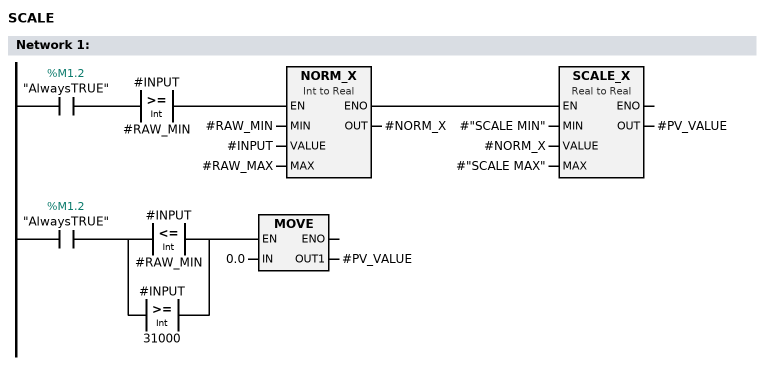
   RUNG wire#powerrail
      Contact( "AlwaysTRUE" )
      { S7_Templates := "SrcType := Int" } GE_Contact(in1 := #INPUT, in2 := #RAW_MIN)
      { S7_Templates := "[SrcType := Int, DestType := Real]" } Normalize(min := #RAW_MIN, value := #INPUT, max := #RAW_MAX, out => #NORM_X)
      { S7_Templates := "[SrcType := Real, DestType := Real]" } Scale(min := #"SCALE MIN", value := #NORM_X, max := #"SCALE MAX", out => #PV_VALUE)
   END_RUNG
   RUNG wire#powerrail
      Contact( "AlwaysTRUE" )
      wire#w1
      { S7_Templates := "SrcType := Int" } LE_Contact(in1 := #INPUT, in2 := #RAW_MIN)
      wire#w2
      Move(in := 0.0, out1 => #PV_VALUE)
   END_RUNG
   RUNG wire#w1
      { S7_Templates := "SrcType := Int" } GE_Contact(in1 := #INPUT, in2 := 31000)
   END_RUNG wire#w2
   // the same network as SCL:
   IF "AlwaysTRUE" AND (#INPUT >= #RAW_MIN) THEN
       #NORM_X := NORM_X(MIN := #RAW_MIN, VALUE := #INPUT, MAX := #RAW_MAX);
       #PV_VALUE := SCALE_X(MIN := #"SCALE MIN", VALUE := #NORM_X, MAX := #"SCALE MAX");
   END_IF;
   IF "AlwaysTRUE" AND ((#INPUT <= #RAW_MIN) OR (#INPUT >= 31000)) THEN #PV_VALUE := 0.0; END_IF;
END_REGION
END_FUNCTION_BLOCK

FUNCTION "SUB_OUTPUT" : Void   // FC5, LAD
{ S7_Optimized_Access := 'TRUE' }
// stored: SetENOAutomatically false
   VAR_TEMP   // added for the SCL form of the ladder/FBD networks
      _w1 : Bool;
   END_VAR
BEGIN

REGION Network 2: "CENTRIFUGAL_PUMP-1"
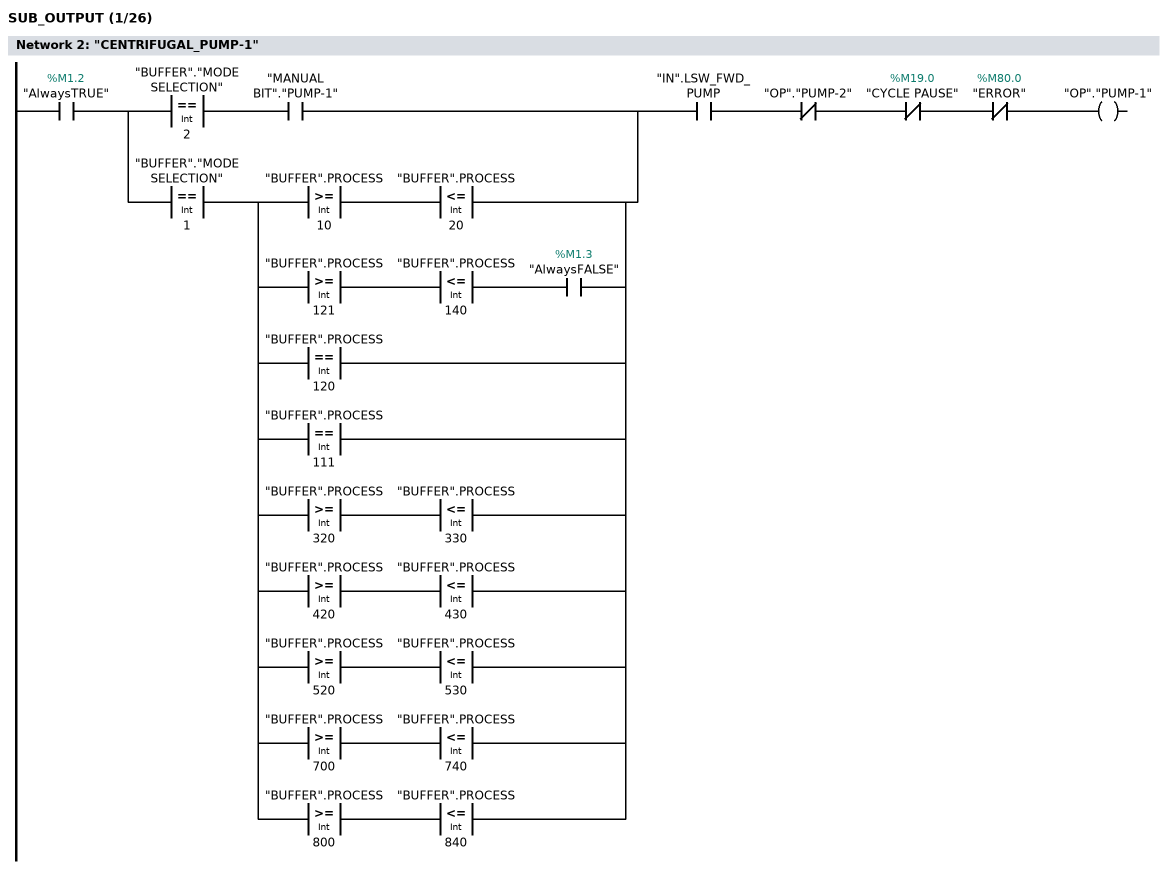
   RUNG wire#powerrail
      Contact( "AlwaysTRUE" )
      wire#w1
      { S7_Templates := "SrcType := Int" } EQ_Contact(in1 := "BUFFER"."MODE SELECTION", in2 := 2)
      Contact( "MANUAL BIT"."PUMP-1" )
      wire#w2
      Contact( "IN".LSW_FWD_PUMP )
      I_Contact( "OP"."PUMP-2" )
      I_Contact( "CYCLE PAUSE" )
      I_Contact( "ERROR" )
      Coil( "OP"."PUMP-1" )
   END_RUNG
   RUNG wire#w1
      { S7_Templates := "SrcType := Int" } EQ_Contact(in1 := "BUFFER"."MODE SELECTION", in2 := 1)
      wire#w3
      { S7_Templates := "SrcType := Int" } GE_Contact(in1 := "BUFFER".PROCESS, in2 := 10)
      { S7_Templates := "SrcType := Int" } LE_Contact(in1 := "BUFFER".PROCESS, in2 := 20)
   END_RUNG wire#w2
   RUNG wire#w3
      { S7_Templates := "SrcType := Int" } GE_Contact(in1 := "BUFFER".PROCESS, in2 := 121)
      { S7_Templates := "SrcType := Int" } LE_Contact(in1 := "BUFFER".PROCESS, in2 := 140)
      Contact( "AlwaysFALSE" )
   END_RUNG wire#w2
   RUNG wire#w3
      { S7_Templates := "SrcType := Int" } EQ_Contact(in1 := "BUFFER".PROCESS, in2 := 120)
   END_RUNG wire#w2
   RUNG wire#w3
      { S7_Templates := "SrcType := Int" } EQ_Contact(in1 := "BUFFER".PROCESS, in2 := 111)
   END_RUNG wire#w2
   RUNG wire#w3
      { S7_Templates := "SrcType := Int" } GE_Contact(in1 := "BUFFER".PROCESS, in2 := 320)
      { S7_Templates := "SrcType := Int" } LE_Contact(in1 := "BUFFER".PROCESS, in2 := 330)
   END_RUNG wire#w2
   RUNG wire#w3
      { S7_Templates := "SrcType := Int" } GE_Contact(in1 := "BUFFER".PROCESS, in2 := 420)
      { S7_Templates := "SrcType := Int" } LE_Contact(in1 := "BUFFER".PROCESS, in2 := 430)
   END_RUNG wire#w2
   RUNG wire#w3
      { S7_Templates := "SrcType := Int" } GE_Contact(in1 := "BUFFER".PROCESS, in2 := 520)
      { S7_Templates := "SrcType := Int" } LE_Contact(in1 := "BUFFER".PROCESS, in2 := 530)
   END_RUNG wire#w2
   RUNG wire#w3
      { S7_Templates := "SrcType := Int" } GE_Contact(in1 := "BUFFER".PROCESS, in2 := 700)
      { S7_Templates := "SrcType := Int" } LE_Contact(in1 := "BUFFER".PROCESS, in2 := 740)
   END_RUNG wire#w2
   RUNG wire#w3
      { S7_Templates := "SrcType := Int" } GE_Contact(in1 := "BUFFER".PROCESS, in2 := 800)
      { S7_Templates := "SrcType := Int" } LE_Contact(in1 := "BUFFER".PROCESS, in2 := 840)
   END_RUNG wire#w2
   // the same network as SCL:
   "OP"."PUMP-1" := "AlwaysTRUE" AND ((("BUFFER"."MODE SELECTION" = 2) AND "MANUAL BIT"."PUMP-1") OR (("BUFFER"."MODE SELECTION" = 1) AND ((("BUFFER".PROCESS >= 10) AND ("BUFFER".PROCESS <= 20)) OR (("BUFFER".PROCESS >= 121) AND ("BUFFER".PROCESS <= 140) AND "AlwaysFALSE") OR ("BUFFER".PROCESS = 120) OR ("BUFFER".PROCESS = 111) OR (("BUFFER".PROCESS >= 320) AND ("BUFFER".PROCESS <= 330)) OR (("BUFFER".PROCESS >= 420) AND ("BUFFER".PROCESS <= 430)) OR (("BUFFER".PROCESS >= 520) AND ("BUFFER".PROCESS <= 530)) OR (("BUFFER".PROCESS >= 700) AND ("BUFFER".PROCESS <= 740)) OR (("BUFFER".PROCESS >= 800) AND ("BUFFER".PROCESS <= 840))))) AND "IN".LSW_FWD_PUMP AND NOT "OP"."PUMP-2" AND NOT "CYCLE PAUSE" AND NOT "ERROR";
END_REGION

REGION Network 3: "CENTRIFUGAL_PUMP-2"
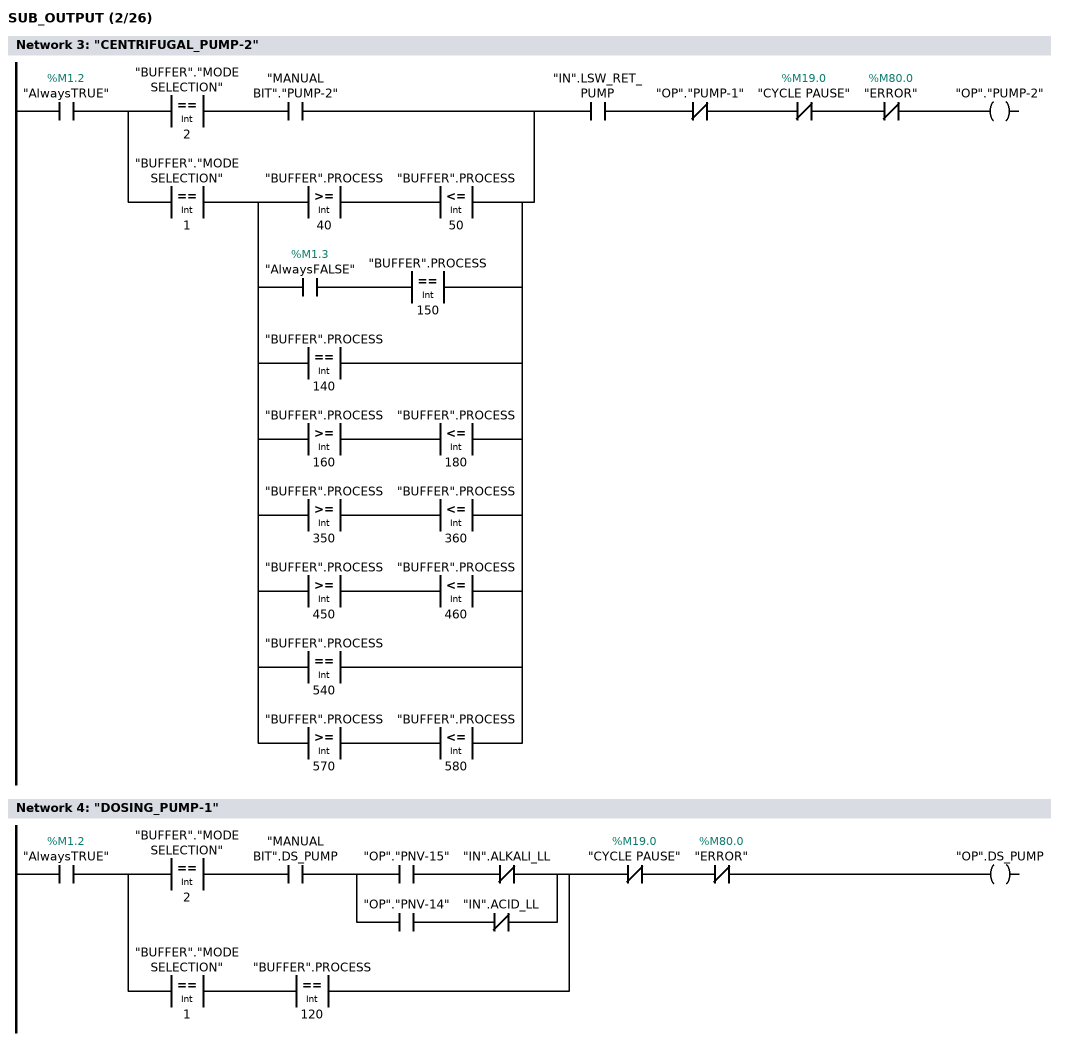
   RUNG wire#powerrail
      Contact( "AlwaysTRUE" )
      wire#w1
      { S7_Templates := "SrcType := Int" } EQ_Contact(in1 := "BUFFER"."MODE SELECTION", in2 := 2)
      Contact( "MANUAL BIT"."PUMP-2" )
      wire#w2
      Contact( "IN".LSW_RET_PUMP )
      I_Contact( "OP"."PUMP-1" )
      I_Contact( "CYCLE PAUSE" )
      I_Contact( "ERROR" )
      Coil( "OP"."PUMP-2" )
   END_RUNG
   RUNG wire#w1
      { S7_Templates := "SrcType := Int" } EQ_Contact(in1 := "BUFFER"."MODE SELECTION", in2 := 1)
      wire#w3
      { S7_Templates := "SrcType := Int" } GE_Contact(in1 := "BUFFER".PROCESS, in2 := 40)
      { S7_Templates := "SrcType := Int" } LE_Contact(in1 := "BUFFER".PROCESS, in2 := 50)
   END_RUNG wire#w2
   RUNG wire#w3
      Contact( "AlwaysFALSE" )
      { S7_Templates := "SrcType := Int" } EQ_Contact(in1 := "BUFFER".PROCESS, in2 := 150)
   END_RUNG wire#w2
   RUNG wire#w3
      { S7_Templates := "SrcType := Int" } EQ_Contact(in1 := "BUFFER".PROCESS, in2 := 140)
   END_RUNG wire#w2
   RUNG wire#w3
      { S7_Templates := "SrcType := Int" } GE_Contact(in1 := "BUFFER".PROCESS, in2 := 160)
      { S7_Templates := "SrcType := Int" } LE_Contact(in1 := "BUFFER".PROCESS, in2 := 180)
   END_RUNG wire#w2
   RUNG wire#w3
      { S7_Templates := "SrcType := Int" } GE_Contact(in1 := "BUFFER".PROCESS, in2 := 350)
      { S7_Templates := "SrcType := Int" } LE_Contact(in1 := "BUFFER".PROCESS, in2 := 360)
   END_RUNG wire#w2
   RUNG wire#w3
      { S7_Templates := "SrcType := Int" } GE_Contact(in1 := "BUFFER".PROCESS, in2 := 450)
      { S7_Templates := "SrcType := Int" } LE_Contact(in1 := "BUFFER".PROCESS, in2 := 460)
   END_RUNG wire#w2
   RUNG wire#w3
      { S7_Templates := "SrcType := Int" } EQ_Contact(in1 := "BUFFER".PROCESS, in2 := 540)
   END_RUNG wire#w2
   RUNG wire#w3
      { S7_Templates := "SrcType := Int" } GE_Contact(in1 := "BUFFER".PROCESS, in2 := 570)
      { S7_Templates := "SrcType := Int" } LE_Contact(in1 := "BUFFER".PROCESS, in2 := 580)
   END_RUNG wire#w2
   // the same network as SCL:
   "OP"."PUMP-2" := "AlwaysTRUE" AND ((("BUFFER"."MODE SELECTION" = 2) AND "MANUAL BIT"."PUMP-2") OR (("BUFFER"."MODE SELECTION" = 1) AND ((("BUFFER".PROCESS >= 40) AND ("BUFFER".PROCESS <= 50)) OR ("AlwaysFALSE" AND ("BUFFER".PROCESS = 150)) OR ("BUFFER".PROCESS = 140) OR (("BUFFER".PROCESS >= 160) AND ("BUFFER".PROCESS <= 180)) OR (("BUFFER".PROCESS >= 350) AND ("BUFFER".PROCESS <= 360)) OR (("BUFFER".PROCESS >= 450) AND ("BUFFER".PROCESS <= 460)) OR ("BUFFER".PROCESS = 540) OR (("BUFFER".PROCESS >= 570) AND ("BUFFER".PROCESS <= 580))))) AND "IN".LSW_RET_PUMP AND NOT "OP"."PUMP-1" AND NOT "CYCLE PAUSE" AND NOT "ERROR";
END_REGION

REGION Network 4: "DOSING_PUMP-1"
   RUNG wire#powerrail
      Contact( "AlwaysTRUE" )
      wire#w1
      { S7_Templates := "SrcType := Int" } EQ_Contact(in1 := "BUFFER"."MODE SELECTION", in2 := 2)
      Contact( "MANUAL BIT".DS_PUMP )
      wire#w2
      Contact( "OP"."PNV-15" )
      I_Contact( "IN".ALKALI_LL )
      wire#w3
      I_Contact( "CYCLE PAUSE" )
      I_Contact( "ERROR" )
      Coil( "OP".DS_PUMP )
   END_RUNG
   RUNG wire#w2
      Contact( "OP"."PNV-14" )
      I_Contact( "IN".ACID_LL )
   END_RUNG wire#w3
   RUNG wire#w1
      { S7_Templates := "SrcType := Int" } EQ_Contact(in1 := "BUFFER"."MODE SELECTION", in2 := 1)
      { S7_Templates := "SrcType := Int" } EQ_Contact(in1 := "BUFFER".PROCESS, in2 := 120)
   END_RUNG wire#w3
   // the same network as SCL:
   "OP".DS_PUMP := "AlwaysTRUE" AND ((("BUFFER"."MODE SELECTION" = 2) AND "MANUAL BIT".DS_PUMP AND (("OP"."PNV-15" AND NOT "IN".ALKALI_LL) OR ("OP"."PNV-14" AND NOT "IN".ACID_LL))) OR (("BUFFER"."MODE SELECTION" = 1) AND ("BUFFER".PROCESS = 120))) AND NOT "CYCLE PAUSE" AND NOT "ERROR";
END_REGION

REGION Network 5: "PNEUMATIC_VALVE-1" (PBFV-1) MFG1- SUGAR
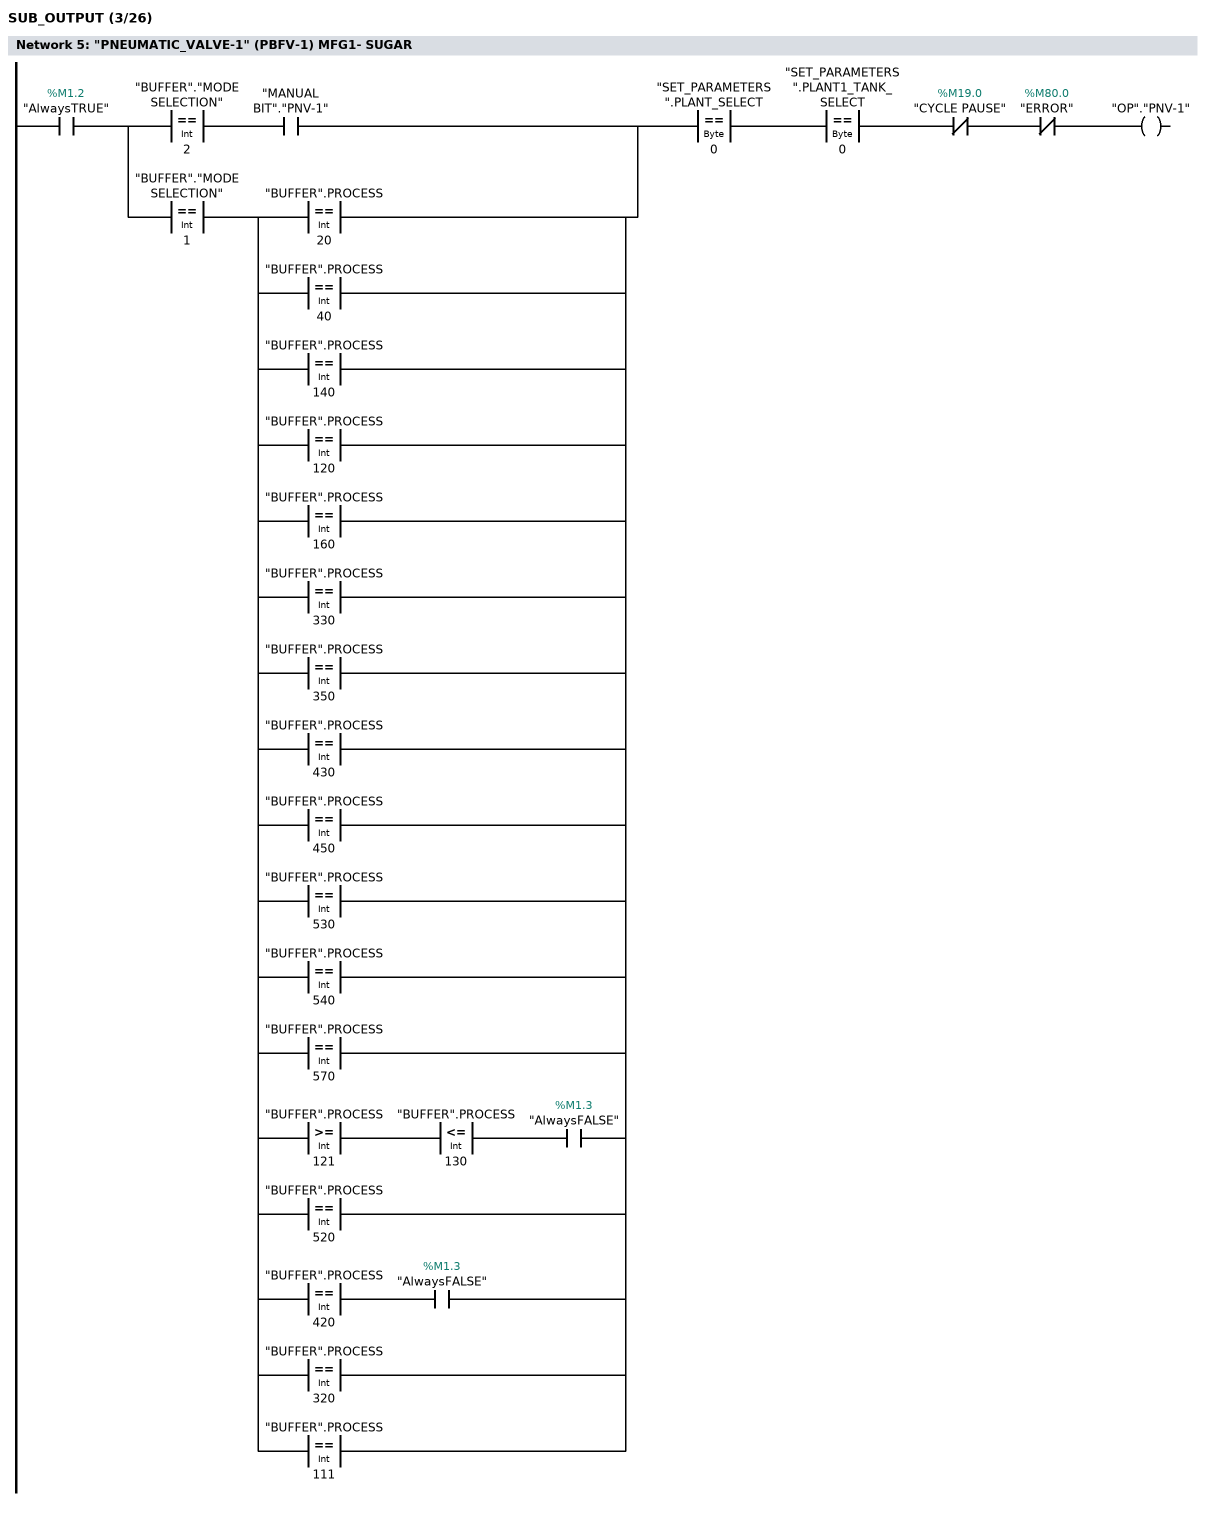
   RUNG wire#powerrail
      Contact( "AlwaysTRUE" )
      wire#w1
      { S7_Templates := "SrcType := Int" } EQ_Contact(in1 := "BUFFER"."MODE SELECTION", in2 := 2)
      Contact( "MANUAL BIT"."PNV-1" )
      wire#w2
      { S7_Templates := "SrcType := Byte" } EQ_Contact(in1 := "SET_PARAMETERS".PLANT_SELECT, in2 := 0)
      { S7_Templates := "SrcType := Byte" } EQ_Contact(in1 := "SET_PARAMETERS".PLANT1_TANK_SELECT, in2 := 0)
      I_Contact( "CYCLE PAUSE" )
      I_Contact( "ERROR" )
      Coil( "OP"."PNV-1" )
   END_RUNG
   RUNG wire#w1
      { S7_Templates := "SrcType := Int" } EQ_Contact(in1 := "BUFFER"."MODE SELECTION", in2 := 1)
      wire#w3
      { S7_Templates := "SrcType := Int" } EQ_Contact(in1 := "BUFFER".PROCESS, in2 := 20)
   END_RUNG wire#w2
   RUNG wire#w3
      { S7_Templates := "SrcType := Int" } EQ_Contact(in1 := "BUFFER".PROCESS, in2 := 40)
   END_RUNG wire#w2
   RUNG wire#w3
      { S7_Templates := "SrcType := Int" } EQ_Contact(in1 := "BUFFER".PROCESS, in2 := 140)
   END_RUNG wire#w2
   RUNG wire#w3
      { S7_Templates := "SrcType := Int" } EQ_Contact(in1 := "BUFFER".PROCESS, in2 := 120)
   END_RUNG wire#w2
   RUNG wire#w3
      { S7_Templates := "SrcType := Int" } EQ_Contact(in1 := "BUFFER".PROCESS, in2 := 160)
   END_RUNG wire#w2
   RUNG wire#w3
      { S7_Templates := "SrcType := Int" } EQ_Contact(in1 := "BUFFER".PROCESS, in2 := 330)
   END_RUNG wire#w2
   RUNG wire#w3
      { S7_Templates := "SrcType := Int" } EQ_Contact(in1 := "BUFFER".PROCESS, in2 := 350)
   END_RUNG wire#w2
   RUNG wire#w3
      { S7_Templates := "SrcType := Int" } EQ_Contact(in1 := "BUFFER".PROCESS, in2 := 430)
   END_RUNG wire#w2
   RUNG wire#w3
      { S7_Templates := "SrcType := Int" } EQ_Contact(in1 := "BUFFER".PROCESS, in2 := 450)
   END_RUNG wire#w2
   RUNG wire#w3
      { S7_Templates := "SrcType := Int" } EQ_Contact(in1 := "BUFFER".PROCESS, in2 := 530)
   END_RUNG wire#w2
   RUNG wire#w3
      { S7_Templates := "SrcType := Int" } EQ_Contact(in1 := "BUFFER".PROCESS, in2 := 540)
   END_RUNG wire#w2
   RUNG wire#w3
      { S7_Templates := "SrcType := Int" } EQ_Contact(in1 := "BUFFER".PROCESS, in2 := 570)
   END_RUNG wire#w2
   RUNG wire#w3
      { S7_Templates := "SrcType := Int" } GE_Contact(in1 := "BUFFER".PROCESS, in2 := 121)
      { S7_Templates := "SrcType := Int" } LE_Contact(in1 := "BUFFER".PROCESS, in2 := 130)
      Contact( "AlwaysFALSE" )
   END_RUNG wire#w2
   RUNG wire#w3
      { S7_Templates := "SrcType := Int" } EQ_Contact(in1 := "BUFFER".PROCESS, in2 := 520)
   END_RUNG wire#w2
   RUNG wire#w3
      { S7_Templates := "SrcType := Int" } EQ_Contact(in1 := "BUFFER".PROCESS, in2 := 420)
      Contact( "AlwaysFALSE" )
   END_RUNG wire#w2
   RUNG wire#w3
      { S7_Templates := "SrcType := Int" } EQ_Contact(in1 := "BUFFER".PROCESS, in2 := 320)
   END_RUNG wire#w2
   RUNG wire#w3
      { S7_Templates := "SrcType := Int" } EQ_Contact(in1 := "BUFFER".PROCESS, in2 := 111)
   END_RUNG wire#w2
   // the same network as SCL:
   "OP"."PNV-1" := "AlwaysTRUE" AND ((("BUFFER"."MODE SELECTION" = 2) AND "MANUAL BIT"."PNV-1") OR (("BUFFER"."MODE SELECTION" = 1) AND (("BUFFER".PROCESS = 20) OR ("BUFFER".PROCESS = 40) OR ("BUFFER".PROCESS = 140) OR ("BUFFER".PROCESS = 120) OR ("BUFFER".PROCESS = 160) OR ("BUFFER".PROCESS = 330) OR ("BUFFER".PROCESS = 350) OR ("BUFFER".PROCESS = 430) OR ("BUFFER".PROCESS = 450) OR ("BUFFER".PROCESS = 530) OR ("BUFFER".PROCESS = 540) OR ("BUFFER".PROCESS = 570) OR (("BUFFER".PROCESS >= 121) AND ("BUFFER".PROCESS <= 130) AND "AlwaysFALSE") OR ("BUFFER".PROCESS = 520) OR (("BUFFER".PROCESS = 420) AND "AlwaysFALSE") OR ("BUFFER".PROCESS = 320) OR ("BUFFER".PROCESS = 111)))) AND ("SET_PARAMETERS".PLANT_SELECT = 0) AND ("SET_PARAMETERS".PLANT1_TANK_SELECT = 0) AND NOT "CYCLE PAUSE" AND NOT "ERROR";
END_REGION

REGION Network 6: "PNEUMATIC_VALVE-2" (PBFV-2) MFG1- MFG
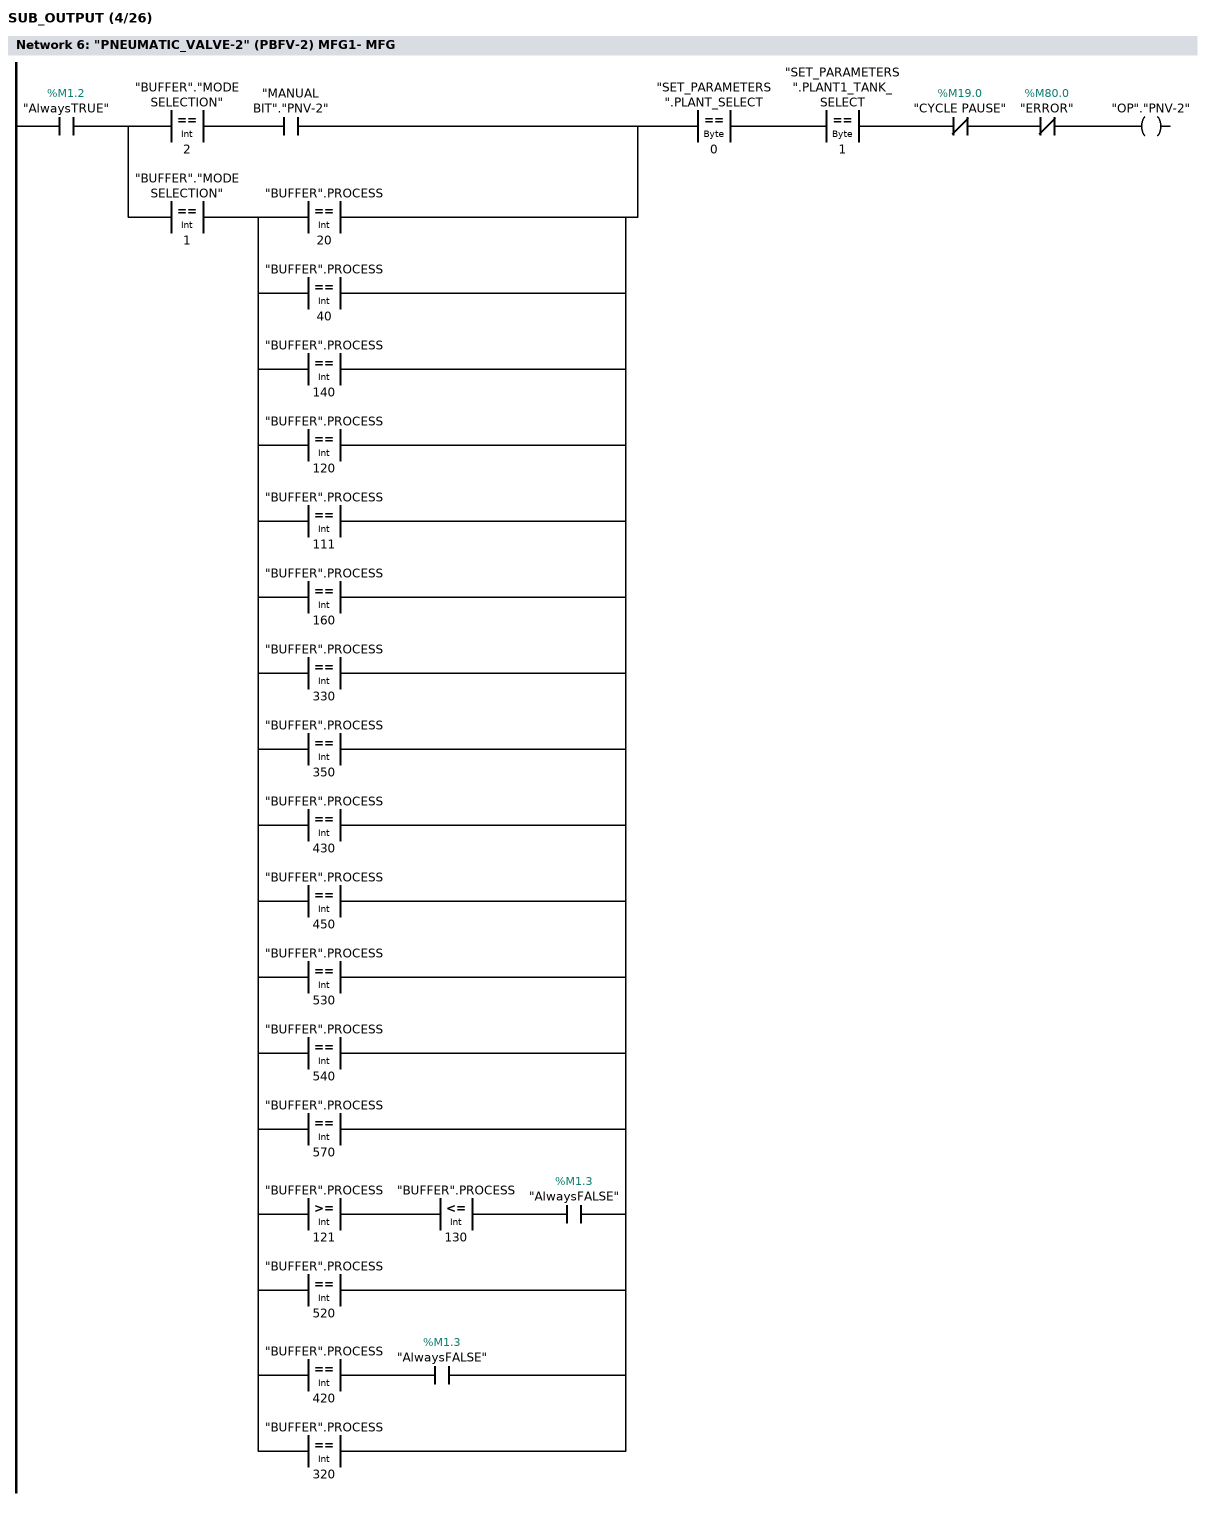
   RUNG wire#powerrail
      Contact( "AlwaysTRUE" )
      wire#w1
      { S7_Templates := "SrcType := Int" } EQ_Contact(in1 := "BUFFER"."MODE SELECTION", in2 := 2)
      Contact( "MANUAL BIT"."PNV-2" )
      wire#w2
      { S7_Templates := "SrcType := Byte" } EQ_Contact(in1 := "SET_PARAMETERS".PLANT_SELECT, in2 := 0)
      { S7_Templates := "SrcType := Byte" } EQ_Contact(in1 := "SET_PARAMETERS".PLANT1_TANK_SELECT, in2 := 1)
      I_Contact( "CYCLE PAUSE" )
      I_Contact( "ERROR" )
      Coil( "OP"."PNV-2" )
   END_RUNG
   RUNG wire#w1
      { S7_Templates := "SrcType := Int" } EQ_Contact(in1 := "BUFFER"."MODE SELECTION", in2 := 1)
      wire#w3
      { S7_Templates := "SrcType := Int" } EQ_Contact(in1 := "BUFFER".PROCESS, in2 := 20)
   END_RUNG wire#w2
   RUNG wire#w3
      { S7_Templates := "SrcType := Int" } EQ_Contact(in1 := "BUFFER".PROCESS, in2 := 40)
   END_RUNG wire#w2
   RUNG wire#w3
      { S7_Templates := "SrcType := Int" } EQ_Contact(in1 := "BUFFER".PROCESS, in2 := 140)
   END_RUNG wire#w2
   RUNG wire#w3
      { S7_Templates := "SrcType := Int" } EQ_Contact(in1 := "BUFFER".PROCESS, in2 := 120)
   END_RUNG wire#w2
   RUNG wire#w3
      { S7_Templates := "SrcType := Int" } EQ_Contact(in1 := "BUFFER".PROCESS, in2 := 111)
   END_RUNG wire#w2
   RUNG wire#w3
      { S7_Templates := "SrcType := Int" } EQ_Contact(in1 := "BUFFER".PROCESS, in2 := 160)
   END_RUNG wire#w2
   RUNG wire#w3
      { S7_Templates := "SrcType := Int" } EQ_Contact(in1 := "BUFFER".PROCESS, in2 := 330)
   END_RUNG wire#w2
   RUNG wire#w3
      { S7_Templates := "SrcType := Int" } EQ_Contact(in1 := "BUFFER".PROCESS, in2 := 350)
   END_RUNG wire#w2
   RUNG wire#w3
      { S7_Templates := "SrcType := Int" } EQ_Contact(in1 := "BUFFER".PROCESS, in2 := 430)
   END_RUNG wire#w2
   RUNG wire#w3
      { S7_Templates := "SrcType := Int" } EQ_Contact(in1 := "BUFFER".PROCESS, in2 := 450)
   END_RUNG wire#w2
   RUNG wire#w3
      { S7_Templates := "SrcType := Int" } EQ_Contact(in1 := "BUFFER".PROCESS, in2 := 530)
   END_RUNG wire#w2
   RUNG wire#w3
      { S7_Templates := "SrcType := Int" } EQ_Contact(in1 := "BUFFER".PROCESS, in2 := 540)
   END_RUNG wire#w2
   RUNG wire#w3
      { S7_Templates := "SrcType := Int" } EQ_Contact(in1 := "BUFFER".PROCESS, in2 := 570)
   END_RUNG wire#w2
   RUNG wire#w3
      { S7_Templates := "SrcType := Int" } GE_Contact(in1 := "BUFFER".PROCESS, in2 := 121)
      { S7_Templates := "SrcType := Int" } LE_Contact(in1 := "BUFFER".PROCESS, in2 := 130)
      Contact( "AlwaysFALSE" )
   END_RUNG wire#w2
   RUNG wire#w3
      { S7_Templates := "SrcType := Int" } EQ_Contact(in1 := "BUFFER".PROCESS, in2 := 520)
   END_RUNG wire#w2
   RUNG wire#w3
      { S7_Templates := "SrcType := Int" } EQ_Contact(in1 := "BUFFER".PROCESS, in2 := 420)
      Contact( "AlwaysFALSE" )
   END_RUNG wire#w2
   RUNG wire#w3
      { S7_Templates := "SrcType := Int" } EQ_Contact(in1 := "BUFFER".PROCESS, in2 := 320)
   END_RUNG wire#w2
   // the same network as SCL:
   "OP"."PNV-2" := "AlwaysTRUE" AND ((("BUFFER"."MODE SELECTION" = 2) AND "MANUAL BIT"."PNV-2") OR (("BUFFER"."MODE SELECTION" = 1) AND (("BUFFER".PROCESS = 20) OR ("BUFFER".PROCESS = 40) OR ("BUFFER".PROCESS = 140) OR ("BUFFER".PROCESS = 120) OR ("BUFFER".PROCESS = 111) OR ("BUFFER".PROCESS = 160) OR ("BUFFER".PROCESS = 330) OR ("BUFFER".PROCESS = 350) OR ("BUFFER".PROCESS = 430) OR ("BUFFER".PROCESS = 450) OR ("BUFFER".PROCESS = 530) OR ("BUFFER".PROCESS = 540) OR ("BUFFER".PROCESS = 570) OR (("BUFFER".PROCESS >= 121) AND ("BUFFER".PROCESS <= 130) AND "AlwaysFALSE") OR ("BUFFER".PROCESS = 520) OR (("BUFFER".PROCESS = 420) AND "AlwaysFALSE") OR ("BUFFER".PROCESS = 320)))) AND ("SET_PARAMETERS".PLANT_SELECT = 0) AND ("SET_PARAMETERS".PLANT1_TANK_SELECT = 1) AND NOT "CYCLE PAUSE" AND NOT "ERROR";
END_REGION

REGION Network 7: "PNEUMATIC_VALVE-3" (PBFV-3)
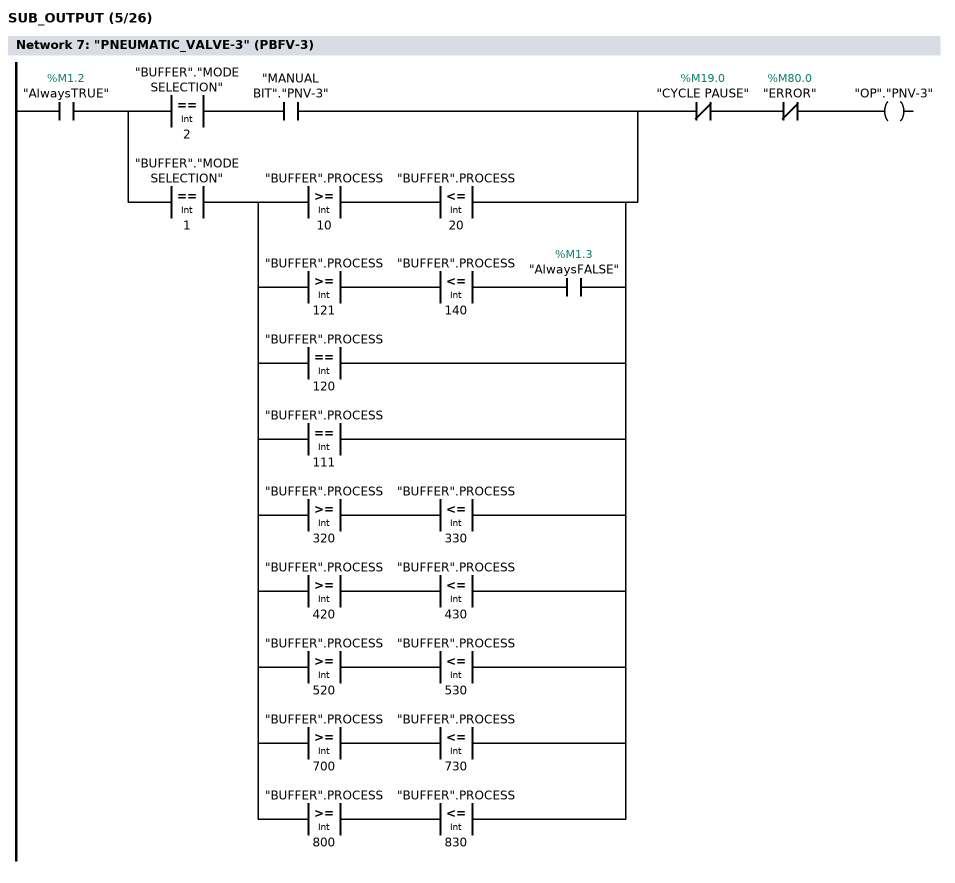
   RUNG wire#powerrail
      Contact( "AlwaysTRUE" )
      wire#w1
      { S7_Templates := "SrcType := Int" } EQ_Contact(in1 := "BUFFER"."MODE SELECTION", in2 := 2)
      Contact( "MANUAL BIT"."PNV-3" )
      wire#w2
      I_Contact( "CYCLE PAUSE" )
      I_Contact( "ERROR" )
      Coil( "OP"."PNV-3" )
   END_RUNG
   RUNG wire#w1
      { S7_Templates := "SrcType := Int" } EQ_Contact(in1 := "BUFFER"."MODE SELECTION", in2 := 1)
      wire#w3
      { S7_Templates := "SrcType := Int" } GE_Contact(in1 := "BUFFER".PROCESS, in2 := 10)
      { S7_Templates := "SrcType := Int" } LE_Contact(in1 := "BUFFER".PROCESS, in2 := 20)
   END_RUNG wire#w2
   RUNG wire#w3
      { S7_Templates := "SrcType := Int" } GE_Contact(in1 := "BUFFER".PROCESS, in2 := 121)
      { S7_Templates := "SrcType := Int" } LE_Contact(in1 := "BUFFER".PROCESS, in2 := 140)
      Contact( "AlwaysFALSE" )
   END_RUNG wire#w2
   RUNG wire#w3
      { S7_Templates := "SrcType := Int" } EQ_Contact(in1 := "BUFFER".PROCESS, in2 := 120)
   END_RUNG wire#w2
   RUNG wire#w3
      { S7_Templates := "SrcType := Int" } EQ_Contact(in1 := "BUFFER".PROCESS, in2 := 111)
   END_RUNG wire#w2
   RUNG wire#w3
      { S7_Templates := "SrcType := Int" } GE_Contact(in1 := "BUFFER".PROCESS, in2 := 320)
      { S7_Templates := "SrcType := Int" } LE_Contact(in1 := "BUFFER".PROCESS, in2 := 330)
   END_RUNG wire#w2
   RUNG wire#w3
      { S7_Templates := "SrcType := Int" } GE_Contact(in1 := "BUFFER".PROCESS, in2 := 420)
      { S7_Templates := "SrcType := Int" } LE_Contact(in1 := "BUFFER".PROCESS, in2 := 430)
   END_RUNG wire#w2
   RUNG wire#w3
      { S7_Templates := "SrcType := Int" } GE_Contact(in1 := "BUFFER".PROCESS, in2 := 520)
      { S7_Templates := "SrcType := Int" } LE_Contact(in1 := "BUFFER".PROCESS, in2 := 530)
   END_RUNG wire#w2
   RUNG wire#w3
      { S7_Templates := "SrcType := Int" } GE_Contact(in1 := "BUFFER".PROCESS, in2 := 700)
      { S7_Templates := "SrcType := Int" } LE_Contact(in1 := "BUFFER".PROCESS, in2 := 730)
   END_RUNG wire#w2
   RUNG wire#w3
      { S7_Templates := "SrcType := Int" } GE_Contact(in1 := "BUFFER".PROCESS, in2 := 800)
      { S7_Templates := "SrcType := Int" } LE_Contact(in1 := "BUFFER".PROCESS, in2 := 830)
   END_RUNG wire#w2
   // the same network as SCL:
   "OP"."PNV-3" := "AlwaysTRUE" AND ((("BUFFER"."MODE SELECTION" = 2) AND "MANUAL BIT"."PNV-3") OR (("BUFFER"."MODE SELECTION" = 1) AND ((("BUFFER".PROCESS >= 10) AND ("BUFFER".PROCESS <= 20)) OR (("BUFFER".PROCESS >= 121) AND ("BUFFER".PROCESS <= 140) AND "AlwaysFALSE") OR ("BUFFER".PROCESS = 120) OR ("BUFFER".PROCESS = 111) OR (("BUFFER".PROCESS >= 320) AND ("BUFFER".PROCESS <= 330)) OR (("BUFFER".PROCESS >= 420) AND ("BUFFER".PROCESS <= 430)) OR (("BUFFER".PROCESS >= 520) AND ("BUFFER".PROCESS <= 530)) OR (("BUFFER".PROCESS >= 700) AND ("BUFFER".PROCESS <= 730)) OR (("BUFFER".PROCESS >= 800) AND ("BUFFER".PROCESS <= 830))))) AND NOT "CYCLE PAUSE" AND NOT "ERROR";
END_REGION

REGION Network 8: "PNEUMATIC_VALVE-4" (PBFV-4)
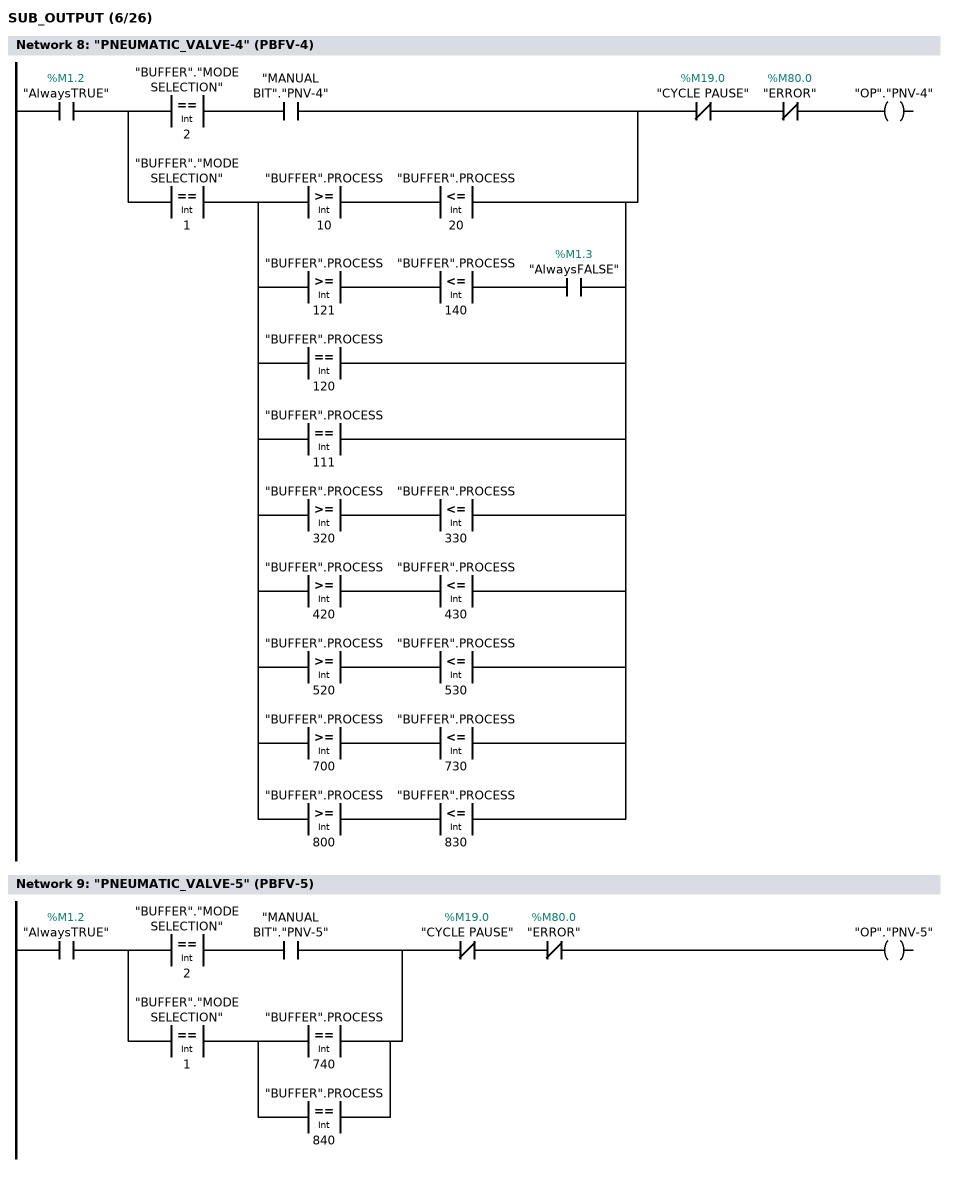
   RUNG wire#powerrail
      Contact( "AlwaysTRUE" )
      wire#w1
      { S7_Templates := "SrcType := Int" } EQ_Contact(in1 := "BUFFER"."MODE SELECTION", in2 := 2)
      Contact( "MANUAL BIT"."PNV-4" )
      wire#w2
      I_Contact( "CYCLE PAUSE" )
      I_Contact( "ERROR" )
      Coil( "OP"."PNV-4" )
   END_RUNG
   RUNG wire#w1
      { S7_Templates := "SrcType := Int" } EQ_Contact(in1 := "BUFFER"."MODE SELECTION", in2 := 1)
      wire#w3
      { S7_Templates := "SrcType := Int" } GE_Contact(in1 := "BUFFER".PROCESS, in2 := 10)
      { S7_Templates := "SrcType := Int" } LE_Contact(in1 := "BUFFER".PROCESS, in2 := 20)
   END_RUNG wire#w2
   RUNG wire#w3
      { S7_Templates := "SrcType := Int" } GE_Contact(in1 := "BUFFER".PROCESS, in2 := 121)
      { S7_Templates := "SrcType := Int" } LE_Contact(in1 := "BUFFER".PROCESS, in2 := 140)
      Contact( "AlwaysFALSE" )
   END_RUNG wire#w2
   RUNG wire#w3
      { S7_Templates := "SrcType := Int" } EQ_Contact(in1 := "BUFFER".PROCESS, in2 := 120)
   END_RUNG wire#w2
   RUNG wire#w3
      { S7_Templates := "SrcType := Int" } EQ_Contact(in1 := "BUFFER".PROCESS, in2 := 111)
   END_RUNG wire#w2
   RUNG wire#w3
      { S7_Templates := "SrcType := Int" } GE_Contact(in1 := "BUFFER".PROCESS, in2 := 320)
      { S7_Templates := "SrcType := Int" } LE_Contact(in1 := "BUFFER".PROCESS, in2 := 330)
   END_RUNG wire#w2
   RUNG wire#w3
      { S7_Templates := "SrcType := Int" } GE_Contact(in1 := "BUFFER".PROCESS, in2 := 420)
      { S7_Templates := "SrcType := Int" } LE_Contact(in1 := "BUFFER".PROCESS, in2 := 430)
   END_RUNG wire#w2
   RUNG wire#w3
      { S7_Templates := "SrcType := Int" } GE_Contact(in1 := "BUFFER".PROCESS, in2 := 520)
      { S7_Templates := "SrcType := Int" } LE_Contact(in1 := "BUFFER".PROCESS, in2 := 530)
   END_RUNG wire#w2
   RUNG wire#w3
      { S7_Templates := "SrcType := Int" } GE_Contact(in1 := "BUFFER".PROCESS, in2 := 700)
      { S7_Templates := "SrcType := Int" } LE_Contact(in1 := "BUFFER".PROCESS, in2 := 730)
   END_RUNG wire#w2
   RUNG wire#w3
      { S7_Templates := "SrcType := Int" } GE_Contact(in1 := "BUFFER".PROCESS, in2 := 800)
      { S7_Templates := "SrcType := Int" } LE_Contact(in1 := "BUFFER".PROCESS, in2 := 830)
   END_RUNG wire#w2
   // the same network as SCL:
   "OP"."PNV-4" := "AlwaysTRUE" AND ((("BUFFER"."MODE SELECTION" = 2) AND "MANUAL BIT"."PNV-4") OR (("BUFFER"."MODE SELECTION" = 1) AND ((("BUFFER".PROCESS >= 10) AND ("BUFFER".PROCESS <= 20)) OR (("BUFFER".PROCESS >= 121) AND ("BUFFER".PROCESS <= 140) AND "AlwaysFALSE") OR ("BUFFER".PROCESS = 120) OR ("BUFFER".PROCESS = 111) OR (("BUFFER".PROCESS >= 320) AND ("BUFFER".PROCESS <= 330)) OR (("BUFFER".PROCESS >= 420) AND ("BUFFER".PROCESS <= 430)) OR (("BUFFER".PROCESS >= 520) AND ("BUFFER".PROCESS <= 530)) OR (("BUFFER".PROCESS >= 700) AND ("BUFFER".PROCESS <= 730)) OR (("BUFFER".PROCESS >= 800) AND ("BUFFER".PROCESS <= 830))))) AND NOT "CYCLE PAUSE" AND NOT "ERROR";
END_REGION

REGION Network 9: "PNEUMATIC_VALVE-5" (PBFV-5)
   RUNG wire#powerrail
      Contact( "AlwaysTRUE" )
      wire#w1
      { S7_Templates := "SrcType := Int" } EQ_Contact(in1 := "BUFFER"."MODE SELECTION", in2 := 2)
      Contact( "MANUAL BIT"."PNV-5" )
      wire#w2
      I_Contact( "CYCLE PAUSE" )
      I_Contact( "ERROR" )
      Coil( "OP"."PNV-5" )
   END_RUNG
   RUNG wire#w1
      { S7_Templates := "SrcType := Int" } EQ_Contact(in1 := "BUFFER"."MODE SELECTION", in2 := 1)
      wire#w3
      { S7_Templates := "SrcType := Int" } EQ_Contact(in1 := "BUFFER".PROCESS, in2 := 740)
   END_RUNG wire#w2
   RUNG wire#w3
      { S7_Templates := "SrcType := Int" } EQ_Contact(in1 := "BUFFER".PROCESS, in2 := 840)
   END_RUNG wire#w2
   // the same network as SCL:
   "OP"."PNV-5" := "AlwaysTRUE" AND ((("BUFFER"."MODE SELECTION" = 2) AND "MANUAL BIT"."PNV-5") OR (("BUFFER"."MODE SELECTION" = 1) AND (("BUFFER".PROCESS = 740) OR ("BUFFER".PROCESS = 840)))) AND NOT "CYCLE PAUSE" AND NOT "ERROR";
END_REGION

REGION Network 10: "PNEUMATIC_VALVE-6" (PBFV-6)
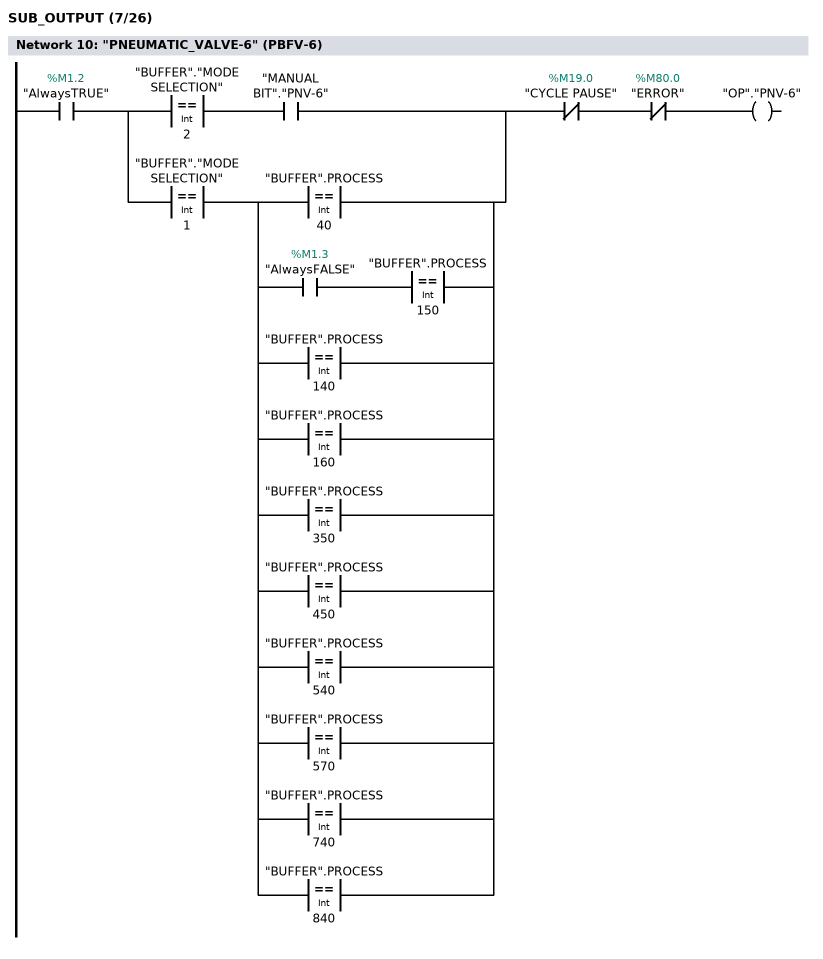
   RUNG wire#powerrail
      Contact( "AlwaysTRUE" )
      wire#w1
      { S7_Templates := "SrcType := Int" } EQ_Contact(in1 := "BUFFER"."MODE SELECTION", in2 := 2)
      Contact( "MANUAL BIT"."PNV-6" )
      wire#w2
      I_Contact( "CYCLE PAUSE" )
      I_Contact( "ERROR" )
      Coil( "OP"."PNV-6" )
   END_RUNG
   RUNG wire#w1
      { S7_Templates := "SrcType := Int" } EQ_Contact(in1 := "BUFFER"."MODE SELECTION", in2 := 1)
      wire#w3
      { S7_Templates := "SrcType := Int" } EQ_Contact(in1 := "BUFFER".PROCESS, in2 := 40)
   END_RUNG wire#w2
   RUNG wire#w3
      Contact( "AlwaysFALSE" )
      { S7_Templates := "SrcType := Int" } EQ_Contact(in1 := "BUFFER".PROCESS, in2 := 150)
   END_RUNG wire#w2
   RUNG wire#w3
      { S7_Templates := "SrcType := Int" } EQ_Contact(in1 := "BUFFER".PROCESS, in2 := 140)
   END_RUNG wire#w2
   RUNG wire#w3
      { S7_Templates := "SrcType := Int" } EQ_Contact(in1 := "BUFFER".PROCESS, in2 := 160)
   END_RUNG wire#w2
   RUNG wire#w3
      { S7_Templates := "SrcType := Int" } EQ_Contact(in1 := "BUFFER".PROCESS, in2 := 350)
   END_RUNG wire#w2
   RUNG wire#w3
      { S7_Templates := "SrcType := Int" } EQ_Contact(in1 := "BUFFER".PROCESS, in2 := 450)
   END_RUNG wire#w2
   RUNG wire#w3
      { S7_Templates := "SrcType := Int" } EQ_Contact(in1 := "BUFFER".PROCESS, in2 := 540)
   END_RUNG wire#w2
   RUNG wire#w3
      { S7_Templates := "SrcType := Int" } EQ_Contact(in1 := "BUFFER".PROCESS, in2 := 570)
   END_RUNG wire#w2
   RUNG wire#w3
      { S7_Templates := "SrcType := Int" } EQ_Contact(in1 := "BUFFER".PROCESS, in2 := 740)
   END_RUNG wire#w2
   RUNG wire#w3
      { S7_Templates := "SrcType := Int" } EQ_Contact(in1 := "BUFFER".PROCESS, in2 := 840)
   END_RUNG wire#w2
   // the same network as SCL:
   "OP"."PNV-6" := "AlwaysTRUE" AND ((("BUFFER"."MODE SELECTION" = 2) AND "MANUAL BIT"."PNV-6") OR (("BUFFER"."MODE SELECTION" = 1) AND (("BUFFER".PROCESS = 40) OR ("AlwaysFALSE" AND ("BUFFER".PROCESS = 150)) OR ("BUFFER".PROCESS = 140) OR ("BUFFER".PROCESS = 160) OR ("BUFFER".PROCESS = 350) OR ("BUFFER".PROCESS = 450) OR ("BUFFER".PROCESS = 540) OR ("BUFFER".PROCESS = 570) OR ("BUFFER".PROCESS = 740) OR ("BUFFER".PROCESS = 840)))) AND NOT "CYCLE PAUSE" AND NOT "ERROR";
END_REGION

REGION Network 11: "PNEUMATIC_VALVE-7" (PBFV-7) SWT RECIRCULATION
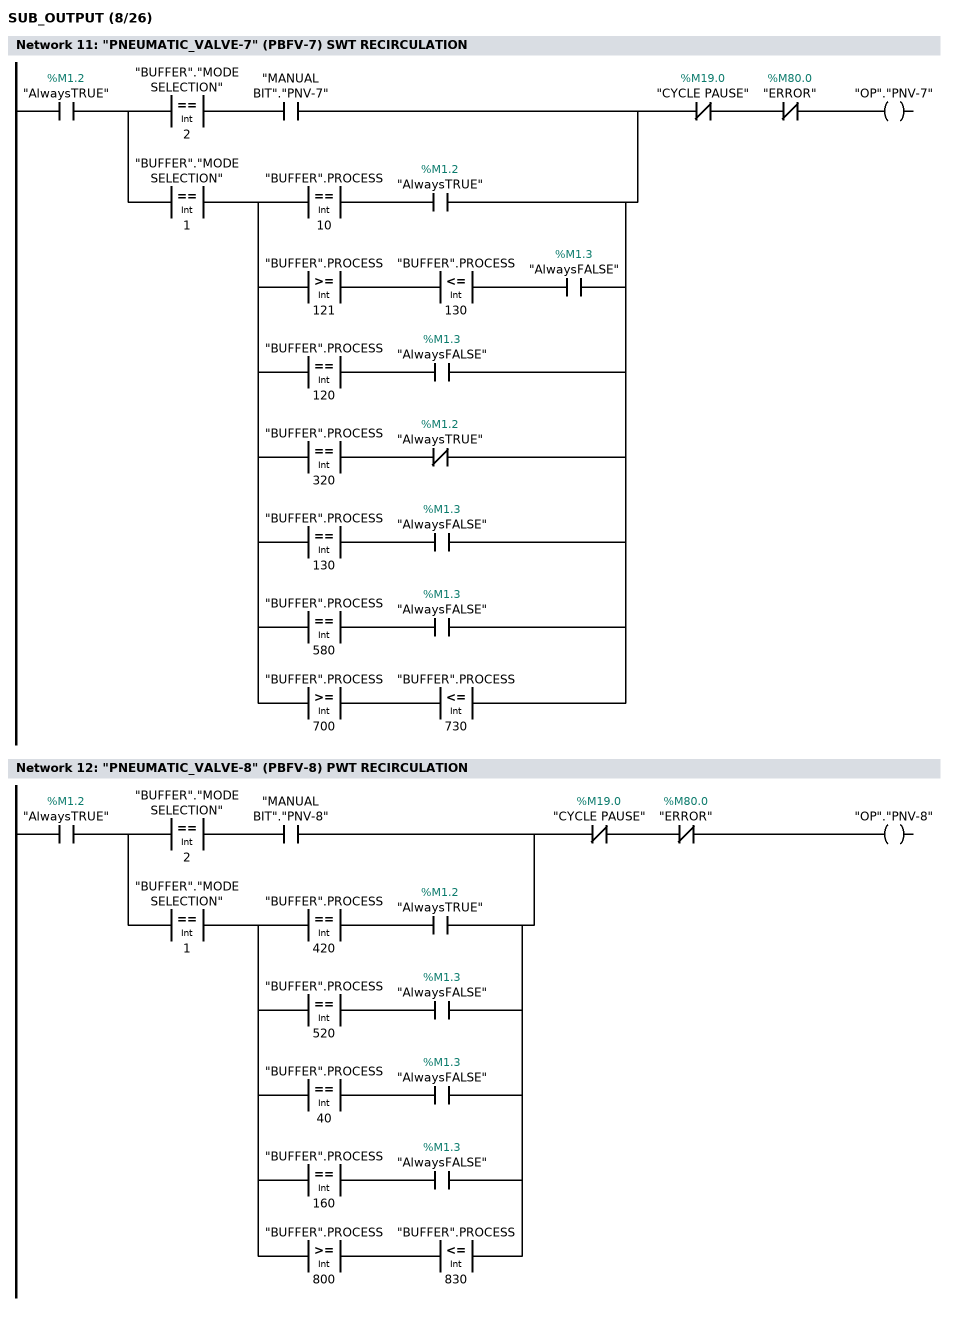
   RUNG wire#powerrail
      Contact( "AlwaysTRUE" )
      wire#w1
      { S7_Templates := "SrcType := Int" } EQ_Contact(in1 := "BUFFER"."MODE SELECTION", in2 := 2)
      Contact( "MANUAL BIT"."PNV-7" )
      wire#w2
      I_Contact( "CYCLE PAUSE" )
      I_Contact( "ERROR" )
      Coil( "OP"."PNV-7" )
   END_RUNG
   RUNG wire#w1
      { S7_Templates := "SrcType := Int" } EQ_Contact(in1 := "BUFFER"."MODE SELECTION", in2 := 1)
      wire#w3
      { S7_Templates := "SrcType := Int" } EQ_Contact(in1 := "BUFFER".PROCESS, in2 := 10)
      Contact( "AlwaysTRUE" )
   END_RUNG wire#w2
   RUNG wire#w3
      { S7_Templates := "SrcType := Int" } GE_Contact(in1 := "BUFFER".PROCESS, in2 := 121)
      { S7_Templates := "SrcType := Int" } LE_Contact(in1 := "BUFFER".PROCESS, in2 := 130)
      Contact( "AlwaysFALSE" )
   END_RUNG wire#w2
   RUNG wire#w3
      { S7_Templates := "SrcType := Int" } EQ_Contact(in1 := "BUFFER".PROCESS, in2 := 120)
      Contact( "AlwaysFALSE" )
   END_RUNG wire#w2
   RUNG wire#w3
      { S7_Templates := "SrcType := Int" } EQ_Contact(in1 := "BUFFER".PROCESS, in2 := 320)
      I_Contact( "AlwaysTRUE" )
   END_RUNG wire#w2
   RUNG wire#w3
      { S7_Templates := "SrcType := Int" } EQ_Contact(in1 := "BUFFER".PROCESS, in2 := 130)
      Contact( "AlwaysFALSE" )
   END_RUNG wire#w2
   RUNG wire#w3
      { S7_Templates := "SrcType := Int" } EQ_Contact(in1 := "BUFFER".PROCESS, in2 := 580)
      Contact( "AlwaysFALSE" )
   END_RUNG wire#w2
   RUNG wire#w3
      { S7_Templates := "SrcType := Int" } GE_Contact(in1 := "BUFFER".PROCESS, in2 := 700)
      { S7_Templates := "SrcType := Int" } LE_Contact(in1 := "BUFFER".PROCESS, in2 := 730)
   END_RUNG wire#w2
   // the same network as SCL:
   "OP"."PNV-7" := "AlwaysTRUE" AND ((("BUFFER"."MODE SELECTION" = 2) AND "MANUAL BIT"."PNV-7") OR (("BUFFER"."MODE SELECTION" = 1) AND ((("BUFFER".PROCESS = 10) AND "AlwaysTRUE") OR (("BUFFER".PROCESS >= 121) AND ("BUFFER".PROCESS <= 130) AND "AlwaysFALSE") OR (("BUFFER".PROCESS = 120) AND "AlwaysFALSE") OR (("BUFFER".PROCESS = 320) AND NOT "AlwaysTRUE") OR (("BUFFER".PROCESS = 130) AND "AlwaysFALSE") OR (("BUFFER".PROCESS = 580) AND "AlwaysFALSE") OR (("BUFFER".PROCESS >= 700) AND ("BUFFER".PROCESS <= 730))))) AND NOT "CYCLE PAUSE" AND NOT "ERROR";
END_REGION

REGION Network 12: "PNEUMATIC_VALVE-8" (PBFV-8) PWT RECIRCULATION
   RUNG wire#powerrail
      Contact( "AlwaysTRUE" )
      wire#w1
      { S7_Templates := "SrcType := Int" } EQ_Contact(in1 := "BUFFER"."MODE SELECTION", in2 := 2)
      Contact( "MANUAL BIT"."PNV-8" )
      wire#w2
      I_Contact( "CYCLE PAUSE" )
      I_Contact( "ERROR" )
      Coil( "OP"."PNV-8" )
   END_RUNG
   RUNG wire#w1
      { S7_Templates := "SrcType := Int" } EQ_Contact(in1 := "BUFFER"."MODE SELECTION", in2 := 1)
      wire#w3
      { S7_Templates := "SrcType := Int" } EQ_Contact(in1 := "BUFFER".PROCESS, in2 := 420)
      Contact( "AlwaysTRUE" )
   END_RUNG wire#w2
   RUNG wire#w3
      { S7_Templates := "SrcType := Int" } EQ_Contact(in1 := "BUFFER".PROCESS, in2 := 520)
      Contact( "AlwaysFALSE" )
   END_RUNG wire#w2
   RUNG wire#w3
      { S7_Templates := "SrcType := Int" } EQ_Contact(in1 := "BUFFER".PROCESS, in2 := 40)
      Contact( "AlwaysFALSE" )
   END_RUNG wire#w2
   RUNG wire#w3
      { S7_Templates := "SrcType := Int" } EQ_Contact(in1 := "BUFFER".PROCESS, in2 := 160)
      Contact( "AlwaysFALSE" )
   END_RUNG wire#w2
   RUNG wire#w3
      { S7_Templates := "SrcType := Int" } GE_Contact(in1 := "BUFFER".PROCESS, in2 := 800)
      { S7_Templates := "SrcType := Int" } LE_Contact(in1 := "BUFFER".PROCESS, in2 := 830)
   END_RUNG wire#w2
   // the same network as SCL:
   "OP"."PNV-8" := "AlwaysTRUE" AND ((("BUFFER"."MODE SELECTION" = 2) AND "MANUAL BIT"."PNV-8") OR (("BUFFER"."MODE SELECTION" = 1) AND ((("BUFFER".PROCESS = 420) AND "AlwaysTRUE") OR (("BUFFER".PROCESS = 520) AND "AlwaysFALSE") OR (("BUFFER".PROCESS = 40) AND "AlwaysFALSE") OR (("BUFFER".PROCESS = 160) AND "AlwaysFALSE") OR (("BUFFER".PROCESS >= 800) AND ("BUFFER".PROCESS <= 830))))) AND NOT "CYCLE PAUSE" AND NOT "ERROR";
END_REGION

REGION Network 13: "PNEUMATIC_VALVE-9" (PBFV-9) MFG-1 - STORAGE1
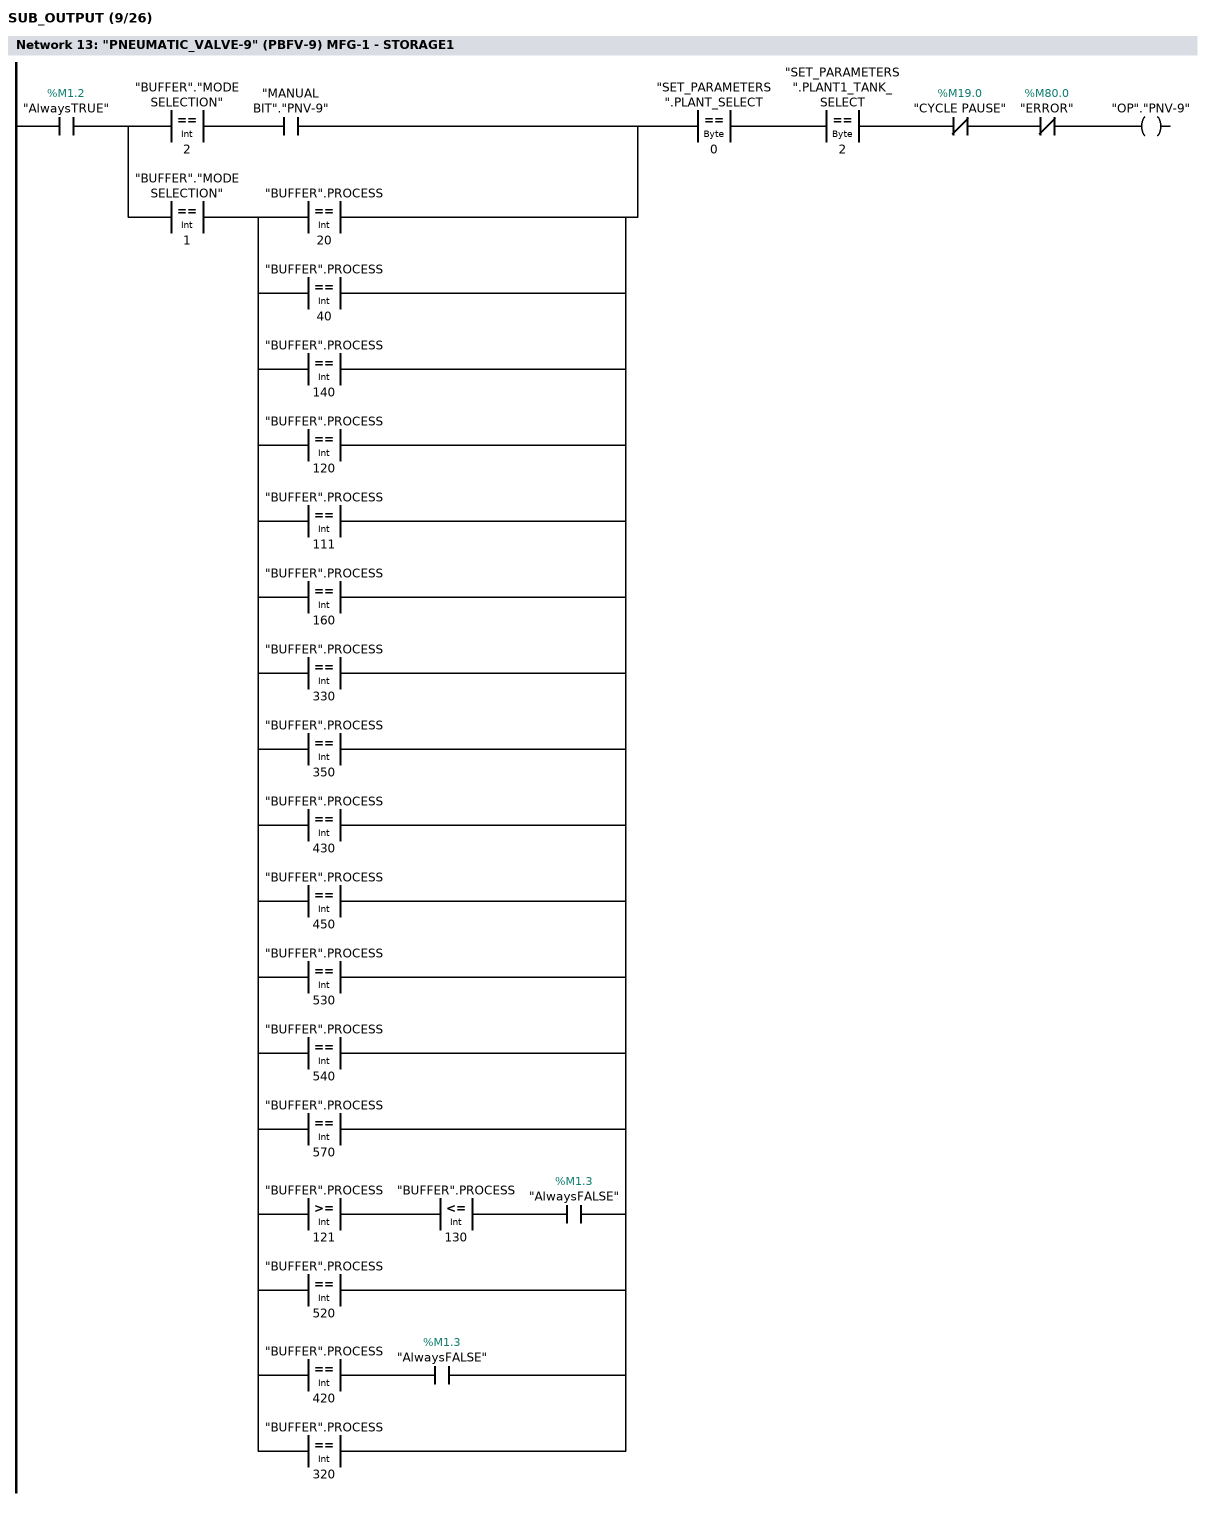
   RUNG wire#powerrail
      Contact( "AlwaysTRUE" )
      wire#w1
      { S7_Templates := "SrcType := Int" } EQ_Contact(in1 := "BUFFER"."MODE SELECTION", in2 := 2)
      Contact( "MANUAL BIT"."PNV-9" )
      wire#w2
      { S7_Templates := "SrcType := Byte" } EQ_Contact(in1 := "SET_PARAMETERS".PLANT_SELECT, in2 := 0)
      { S7_Templates := "SrcType := Byte" } EQ_Contact(in1 := "SET_PARAMETERS".PLANT1_TANK_SELECT, in2 := 2)
      I_Contact( "CYCLE PAUSE" )
      I_Contact( "ERROR" )
      Coil( "OP"."PNV-9" )
   END_RUNG
   RUNG wire#w1
      { S7_Templates := "SrcType := Int" } EQ_Contact(in1 := "BUFFER"."MODE SELECTION", in2 := 1)
      wire#w3
      { S7_Templates := "SrcType := Int" } EQ_Contact(in1 := "BUFFER".PROCESS, in2 := 20)
   END_RUNG wire#w2
   RUNG wire#w3
      { S7_Templates := "SrcType := Int" } EQ_Contact(in1 := "BUFFER".PROCESS, in2 := 40)
   END_RUNG wire#w2
   RUNG wire#w3
      { S7_Templates := "SrcType := Int" } EQ_Contact(in1 := "BUFFER".PROCESS, in2 := 140)
   END_RUNG wire#w2
   RUNG wire#w3
      { S7_Templates := "SrcType := Int" } EQ_Contact(in1 := "BUFFER".PROCESS, in2 := 120)
   END_RUNG wire#w2
   RUNG wire#w3
      { S7_Templates := "SrcType := Int" } EQ_Contact(in1 := "BUFFER".PROCESS, in2 := 111)
   END_RUNG wire#w2
   RUNG wire#w3
      { S7_Templates := "SrcType := Int" } EQ_Contact(in1 := "BUFFER".PROCESS, in2 := 160)
   END_RUNG wire#w2
   RUNG wire#w3
      { S7_Templates := "SrcType := Int" } EQ_Contact(in1 := "BUFFER".PROCESS, in2 := 330)
   END_RUNG wire#w2
   RUNG wire#w3
      { S7_Templates := "SrcType := Int" } EQ_Contact(in1 := "BUFFER".PROCESS, in2 := 350)
   END_RUNG wire#w2
   RUNG wire#w3
      { S7_Templates := "SrcType := Int" } EQ_Contact(in1 := "BUFFER".PROCESS, in2 := 430)
   END_RUNG wire#w2
   RUNG wire#w3
      { S7_Templates := "SrcType := Int" } EQ_Contact(in1 := "BUFFER".PROCESS, in2 := 450)
   END_RUNG wire#w2
   RUNG wire#w3
      { S7_Templates := "SrcType := Int" } EQ_Contact(in1 := "BUFFER".PROCESS, in2 := 530)
   END_RUNG wire#w2
   RUNG wire#w3
      { S7_Templates := "SrcType := Int" } EQ_Contact(in1 := "BUFFER".PROCESS, in2 := 540)
   END_RUNG wire#w2
   RUNG wire#w3
      { S7_Templates := "SrcType := Int" } EQ_Contact(in1 := "BUFFER".PROCESS, in2 := 570)
   END_RUNG wire#w2
   RUNG wire#w3
      { S7_Templates := "SrcType := Int" } GE_Contact(in1 := "BUFFER".PROCESS, in2 := 121)
      { S7_Templates := "SrcType := Int" } LE_Contact(in1 := "BUFFER".PROCESS, in2 := 130)
      Contact( "AlwaysFALSE" )
   END_RUNG wire#w2
   RUNG wire#w3
      { S7_Templates := "SrcType := Int" } EQ_Contact(in1 := "BUFFER".PROCESS, in2 := 520)
   END_RUNG wire#w2
   RUNG wire#w3
      { S7_Templates := "SrcType := Int" } EQ_Contact(in1 := "BUFFER".PROCESS, in2 := 420)
      Contact( "AlwaysFALSE" )
   END_RUNG wire#w2
   RUNG wire#w3
      { S7_Templates := "SrcType := Int" } EQ_Contact(in1 := "BUFFER".PROCESS, in2 := 320)
   END_RUNG wire#w2
   // the same network as SCL:
   "OP"."PNV-9" := "AlwaysTRUE" AND ((("BUFFER"."MODE SELECTION" = 2) AND "MANUAL BIT"."PNV-9") OR (("BUFFER"."MODE SELECTION" = 1) AND (("BUFFER".PROCESS = 20) OR ("BUFFER".PROCESS = 40) OR ("BUFFER".PROCESS = 140) OR ("BUFFER".PROCESS = 120) OR ("BUFFER".PROCESS = 111) OR ("BUFFER".PROCESS = 160) OR ("BUFFER".PROCESS = 330) OR ("BUFFER".PROCESS = 350) OR ("BUFFER".PROCESS = 430) OR ("BUFFER".PROCESS = 450) OR ("BUFFER".PROCESS = 530) OR ("BUFFER".PROCESS = 540) OR ("BUFFER".PROCESS = 570) OR (("BUFFER".PROCESS >= 121) AND ("BUFFER".PROCESS <= 130) AND "AlwaysFALSE") OR ("BUFFER".PROCESS = 520) OR (("BUFFER".PROCESS = 420) AND "AlwaysFALSE") OR ("BUFFER".PROCESS = 320)))) AND ("SET_PARAMETERS".PLANT_SELECT = 0) AND ("SET_PARAMETERS".PLANT1_TANK_SELECT = 2) AND NOT "CYCLE PAUSE" AND NOT "ERROR";
END_REGION

REGION Network 14: "PNEUMATIC_VALVE-10" (PBFV-10) MFG1- STORAGE2
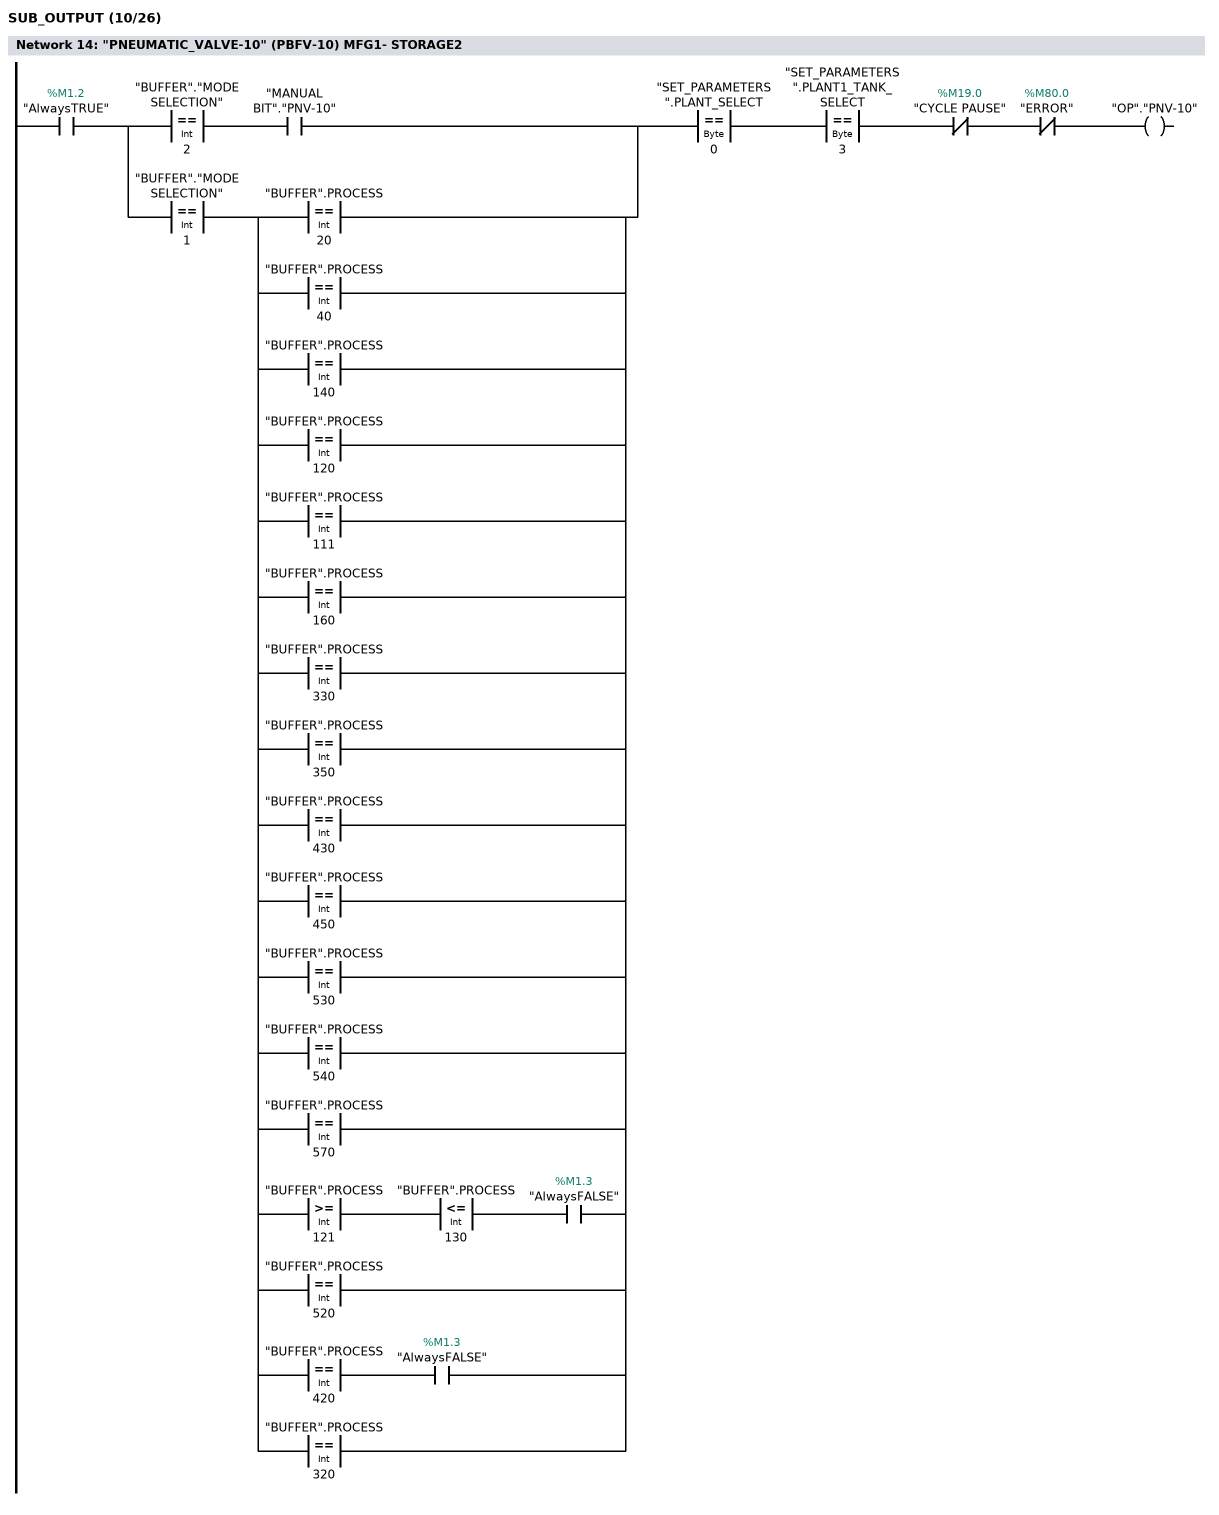
   RUNG wire#powerrail
      Contact( "AlwaysTRUE" )
      wire#w1
      { S7_Templates := "SrcType := Int" } EQ_Contact(in1 := "BUFFER"."MODE SELECTION", in2 := 2)
      Contact( "MANUAL BIT"."PNV-10" )
      wire#w2
      { S7_Templates := "SrcType := Byte" } EQ_Contact(in1 := "SET_PARAMETERS".PLANT_SELECT, in2 := 0)
      { S7_Templates := "SrcType := Byte" } EQ_Contact(in1 := "SET_PARAMETERS".PLANT1_TANK_SELECT, in2 := 3)
      I_Contact( "CYCLE PAUSE" )
      I_Contact( "ERROR" )
      Coil( "OP"."PNV-10" )
   END_RUNG
   RUNG wire#w1
      { S7_Templates := "SrcType := Int" } EQ_Contact(in1 := "BUFFER"."MODE SELECTION", in2 := 1)
      wire#w3
      { S7_Templates := "SrcType := Int" } EQ_Contact(in1 := "BUFFER".PROCESS, in2 := 20)
   END_RUNG wire#w2
   RUNG wire#w3
      { S7_Templates := "SrcType := Int" } EQ_Contact(in1 := "BUFFER".PROCESS, in2 := 40)
   END_RUNG wire#w2
   RUNG wire#w3
      { S7_Templates := "SrcType := Int" } EQ_Contact(in1 := "BUFFER".PROCESS, in2 := 140)
   END_RUNG wire#w2
   RUNG wire#w3
      { S7_Templates := "SrcType := Int" } EQ_Contact(in1 := "BUFFER".PROCESS, in2 := 120)
   END_RUNG wire#w2
   RUNG wire#w3
      { S7_Templates := "SrcType := Int" } EQ_Contact(in1 := "BUFFER".PROCESS, in2 := 111)
   END_RUNG wire#w2
   RUNG wire#w3
      { S7_Templates := "SrcType := Int" } EQ_Contact(in1 := "BUFFER".PROCESS, in2 := 160)
   END_RUNG wire#w2
   RUNG wire#w3
      { S7_Templates := "SrcType := Int" } EQ_Contact(in1 := "BUFFER".PROCESS, in2 := 330)
   END_RUNG wire#w2
   RUNG wire#w3
      { S7_Templates := "SrcType := Int" } EQ_Contact(in1 := "BUFFER".PROCESS, in2 := 350)
   END_RUNG wire#w2
   RUNG wire#w3
      { S7_Templates := "SrcType := Int" } EQ_Contact(in1 := "BUFFER".PROCESS, in2 := 430)
   END_RUNG wire#w2
   RUNG wire#w3
      { S7_Templates := "SrcType := Int" } EQ_Contact(in1 := "BUFFER".PROCESS, in2 := 450)
   END_RUNG wire#w2
   RUNG wire#w3
      { S7_Templates := "SrcType := Int" } EQ_Contact(in1 := "BUFFER".PROCESS, in2 := 530)
   END_RUNG wire#w2
   RUNG wire#w3
      { S7_Templates := "SrcType := Int" } EQ_Contact(in1 := "BUFFER".PROCESS, in2 := 540)
   END_RUNG wire#w2
   RUNG wire#w3
      { S7_Templates := "SrcType := Int" } EQ_Contact(in1 := "BUFFER".PROCESS, in2 := 570)
   END_RUNG wire#w2
   RUNG wire#w3
      { S7_Templates := "SrcType := Int" } GE_Contact(in1 := "BUFFER".PROCESS, in2 := 121)
      { S7_Templates := "SrcType := Int" } LE_Contact(in1 := "BUFFER".PROCESS, in2 := 130)
      Contact( "AlwaysFALSE" )
   END_RUNG wire#w2
   RUNG wire#w3
      { S7_Templates := "SrcType := Int" } EQ_Contact(in1 := "BUFFER".PROCESS, in2 := 520)
   END_RUNG wire#w2
   RUNG wire#w3
      { S7_Templates := "SrcType := Int" } EQ_Contact(in1 := "BUFFER".PROCESS, in2 := 420)
      Contact( "AlwaysFALSE" )
   END_RUNG wire#w2
   RUNG wire#w3
      { S7_Templates := "SrcType := Int" } EQ_Contact(in1 := "BUFFER".PROCESS, in2 := 320)
   END_RUNG wire#w2
   // the same network as SCL:
   "OP"."PNV-10" := "AlwaysTRUE" AND ((("BUFFER"."MODE SELECTION" = 2) AND "MANUAL BIT"."PNV-10") OR (("BUFFER"."MODE SELECTION" = 1) AND (("BUFFER".PROCESS = 20) OR ("BUFFER".PROCESS = 40) OR ("BUFFER".PROCESS = 140) OR ("BUFFER".PROCESS = 120) OR ("BUFFER".PROCESS = 111) OR ("BUFFER".PROCESS = 160) OR ("BUFFER".PROCESS = 330) OR ("BUFFER".PROCESS = 350) OR ("BUFFER".PROCESS = 430) OR ("BUFFER".PROCESS = 450) OR ("BUFFER".PROCESS = 530) OR ("BUFFER".PROCESS = 540) OR ("BUFFER".PROCESS = 570) OR (("BUFFER".PROCESS >= 121) AND ("BUFFER".PROCESS <= 130) AND "AlwaysFALSE") OR ("BUFFER".PROCESS = 520) OR (("BUFFER".PROCESS = 420) AND "AlwaysFALSE") OR ("BUFFER".PROCESS = 320)))) AND ("SET_PARAMETERS".PLANT_SELECT = 0) AND ("SET_PARAMETERS".PLANT1_TANK_SELECT = 3) AND NOT "CYCLE PAUSE" AND NOT "ERROR";
END_REGION

REGION Network 15: "PNEUMATIC_VALVE-11" (PBFV-11)
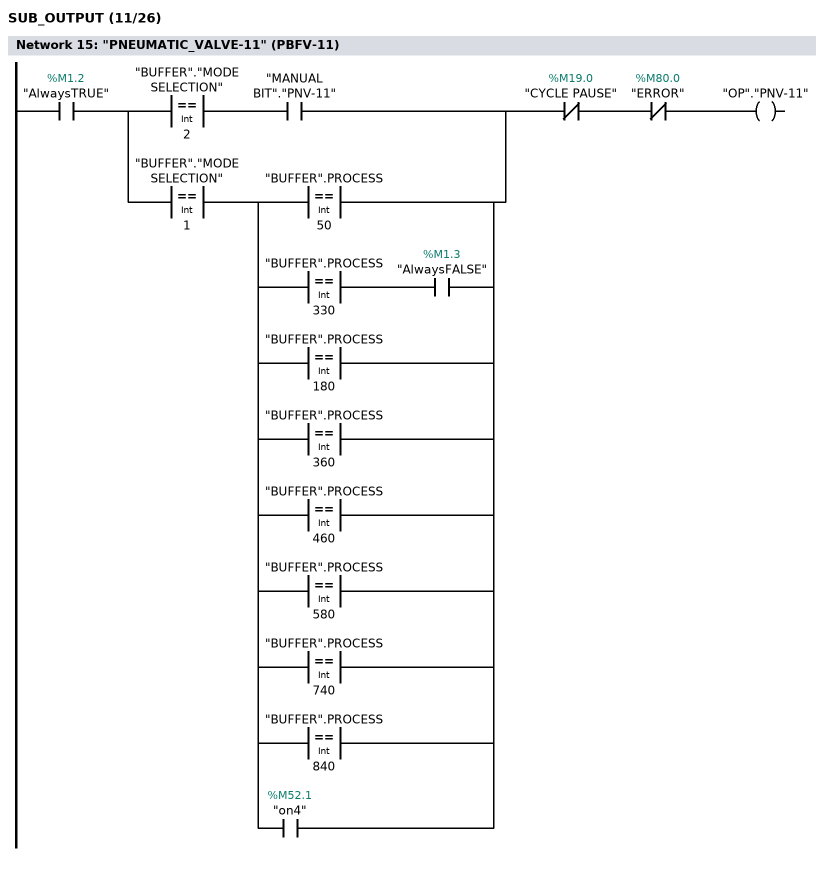
   RUNG wire#powerrail
      Contact( "AlwaysTRUE" )
      wire#w1
      { S7_Templates := "SrcType := Int" } EQ_Contact(in1 := "BUFFER"."MODE SELECTION", in2 := 2)
      Contact( "MANUAL BIT"."PNV-11" )
      wire#w2
      I_Contact( "CYCLE PAUSE" )
      I_Contact( "ERROR" )
      Coil( "OP"."PNV-11" )
   END_RUNG
   RUNG wire#w1
      { S7_Templates := "SrcType := Int" } EQ_Contact(in1 := "BUFFER"."MODE SELECTION", in2 := 1)
      wire#w3
      { S7_Templates := "SrcType := Int" } EQ_Contact(in1 := "BUFFER".PROCESS, in2 := 50)
   END_RUNG wire#w2
   RUNG wire#w3
      { S7_Templates := "SrcType := Int" } EQ_Contact(in1 := "BUFFER".PROCESS, in2 := 330)
      Contact( "AlwaysFALSE" )
   END_RUNG wire#w2
   RUNG wire#w3
      { S7_Templates := "SrcType := Int" } EQ_Contact(in1 := "BUFFER".PROCESS, in2 := 180)
   END_RUNG wire#w2
   RUNG wire#w3
      { S7_Templates := "SrcType := Int" } EQ_Contact(in1 := "BUFFER".PROCESS, in2 := 360)
   END_RUNG wire#w2
   RUNG wire#w3
      { S7_Templates := "SrcType := Int" } EQ_Contact(in1 := "BUFFER".PROCESS, in2 := 460)
   END_RUNG wire#w2
   RUNG wire#w3
      { S7_Templates := "SrcType := Int" } EQ_Contact(in1 := "BUFFER".PROCESS, in2 := 580)
   END_RUNG wire#w2
   RUNG wire#w3
      { S7_Templates := "SrcType := Int" } EQ_Contact(in1 := "BUFFER".PROCESS, in2 := 740)
   END_RUNG wire#w2
   RUNG wire#w3
      { S7_Templates := "SrcType := Int" } EQ_Contact(in1 := "BUFFER".PROCESS, in2 := 840)
   END_RUNG wire#w2
   RUNG wire#w3
      Contact( "on4" )
   END_RUNG wire#w2
   // the same network as SCL:
   "OP"."PNV-11" := "AlwaysTRUE" AND ((("BUFFER"."MODE SELECTION" = 2) AND "MANUAL BIT"."PNV-11") OR (("BUFFER"."MODE SELECTION" = 1) AND (("BUFFER".PROCESS = 50) OR (("BUFFER".PROCESS = 330) AND "AlwaysFALSE") OR ("BUFFER".PROCESS = 180) OR ("BUFFER".PROCESS = 360) OR ("BUFFER".PROCESS = 460) OR ("BUFFER".PROCESS = 580) OR ("BUFFER".PROCESS = 740) OR ("BUFFER".PROCESS = 840) OR "on4"))) AND NOT "CYCLE PAUSE" AND NOT "ERROR";
END_REGION

REGION Network 16: "PNEUMATIC_VALVE-12" (PBFV-12) ONLY MANUAL ACTIVETY NOT USE AUTO LOGIC
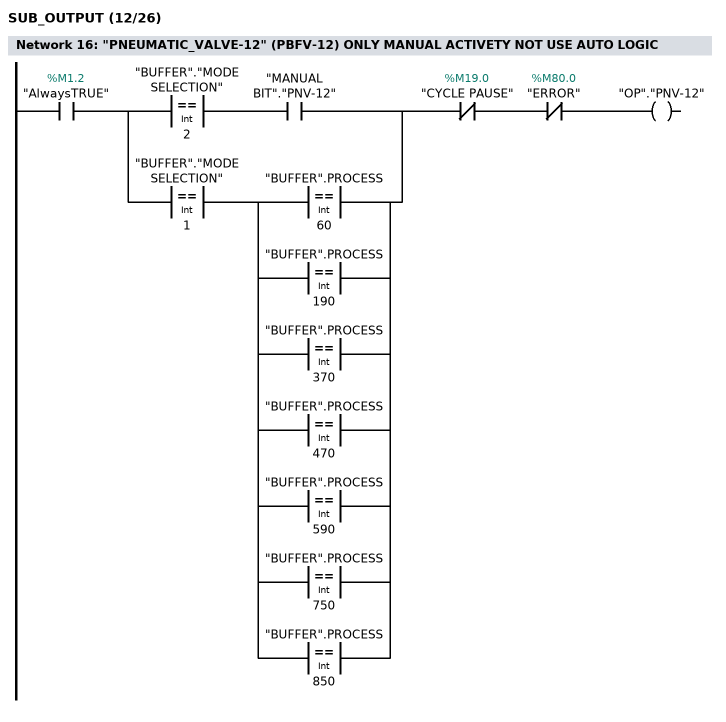
   RUNG wire#powerrail
      Contact( "AlwaysTRUE" )
      wire#w1
      { S7_Templates := "SrcType := Int" } EQ_Contact(in1 := "BUFFER"."MODE SELECTION", in2 := 2)
      Contact( "MANUAL BIT"."PNV-12" )
      wire#w2
      I_Contact( "CYCLE PAUSE" )
      I_Contact( "ERROR" )
      Coil( "OP"."PNV-12" )
   END_RUNG
   RUNG wire#w1
      { S7_Templates := "SrcType := Int" } EQ_Contact(in1 := "BUFFER"."MODE SELECTION", in2 := 1)
      wire#w3
      { S7_Templates := "SrcType := Int" } EQ_Contact(in1 := "BUFFER".PROCESS, in2 := 60)
   END_RUNG wire#w2
   RUNG wire#w3
      { S7_Templates := "SrcType := Int" } EQ_Contact(in1 := "BUFFER".PROCESS, in2 := 190)
   END_RUNG wire#w2
   RUNG wire#w3
      { S7_Templates := "SrcType := Int" } EQ_Contact(in1 := "BUFFER".PROCESS, in2 := 370)
   END_RUNG wire#w2
   RUNG wire#w3
      { S7_Templates := "SrcType := Int" } EQ_Contact(in1 := "BUFFER".PROCESS, in2 := 470)
   END_RUNG wire#w2
   RUNG wire#w3
      { S7_Templates := "SrcType := Int" } EQ_Contact(in1 := "BUFFER".PROCESS, in2 := 590)
   END_RUNG wire#w2
   RUNG wire#w3
      { S7_Templates := "SrcType := Int" } EQ_Contact(in1 := "BUFFER".PROCESS, in2 := 750)
   END_RUNG wire#w2
   RUNG wire#w3
      { S7_Templates := "SrcType := Int" } EQ_Contact(in1 := "BUFFER".PROCESS, in2 := 850)
   END_RUNG wire#w2
   // the same network as SCL:
   "OP"."PNV-12" := "AlwaysTRUE" AND ((("BUFFER"."MODE SELECTION" = 2) AND "MANUAL BIT"."PNV-12") OR (("BUFFER"."MODE SELECTION" = 1) AND (("BUFFER".PROCESS = 60) OR ("BUFFER".PROCESS = 190) OR ("BUFFER".PROCESS = 370) OR ("BUFFER".PROCESS = 470) OR ("BUFFER".PROCESS = 590) OR ("BUFFER".PROCESS = 750) OR ("BUFFER".PROCESS = 850)))) AND NOT "CYCLE PAUSE" AND NOT "ERROR";
END_REGION

REGION Network 17: "PNEUMATIC_VALVE-13" (PBFV-13)
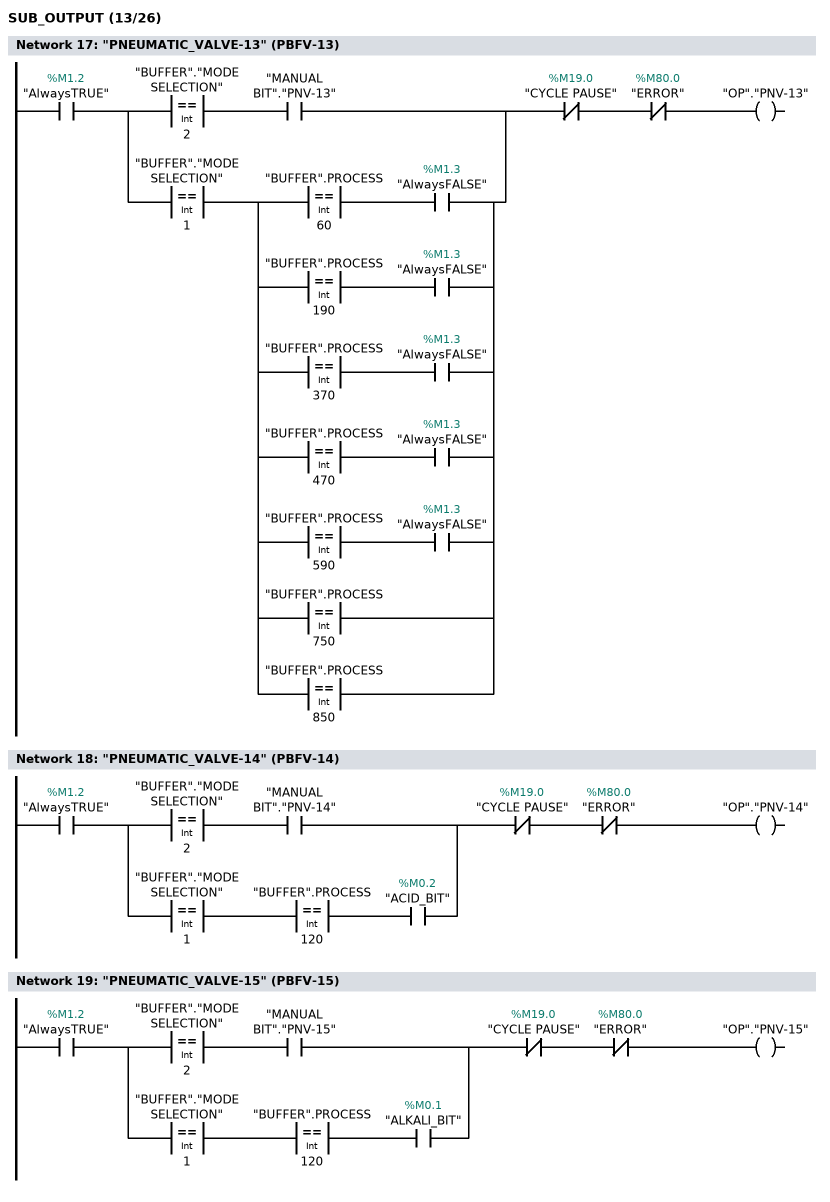
   RUNG wire#powerrail
      Contact( "AlwaysTRUE" )
      wire#w1
      { S7_Templates := "SrcType := Int" } EQ_Contact(in1 := "BUFFER"."MODE SELECTION", in2 := 2)
      Contact( "MANUAL BIT"."PNV-13" )
      wire#w2
      I_Contact( "CYCLE PAUSE" )
      I_Contact( "ERROR" )
      Coil( "OP"."PNV-13" )
   END_RUNG
   RUNG wire#w1
      { S7_Templates := "SrcType := Int" } EQ_Contact(in1 := "BUFFER"."MODE SELECTION", in2 := 1)
      wire#w3
      { S7_Templates := "SrcType := Int" } EQ_Contact(in1 := "BUFFER".PROCESS, in2 := 60)
      Contact( "AlwaysFALSE" )
   END_RUNG wire#w2
   RUNG wire#w3
      { S7_Templates := "SrcType := Int" } EQ_Contact(in1 := "BUFFER".PROCESS, in2 := 190)
      Contact( "AlwaysFALSE" )
   END_RUNG wire#w2
   RUNG wire#w3
      { S7_Templates := "SrcType := Int" } EQ_Contact(in1 := "BUFFER".PROCESS, in2 := 370)
      Contact( "AlwaysFALSE" )
   END_RUNG wire#w2
   RUNG wire#w3
      { S7_Templates := "SrcType := Int" } EQ_Contact(in1 := "BUFFER".PROCESS, in2 := 470)
      Contact( "AlwaysFALSE" )
   END_RUNG wire#w2
   RUNG wire#w3
      { S7_Templates := "SrcType := Int" } EQ_Contact(in1 := "BUFFER".PROCESS, in2 := 590)
      Contact( "AlwaysFALSE" )
   END_RUNG wire#w2
   RUNG wire#w3
      { S7_Templates := "SrcType := Int" } EQ_Contact(in1 := "BUFFER".PROCESS, in2 := 750)
   END_RUNG wire#w2
   RUNG wire#w3
      { S7_Templates := "SrcType := Int" } EQ_Contact(in1 := "BUFFER".PROCESS, in2 := 850)
   END_RUNG wire#w2
   // the same network as SCL:
   "OP"."PNV-13" := "AlwaysTRUE" AND ((("BUFFER"."MODE SELECTION" = 2) AND "MANUAL BIT"."PNV-13") OR (("BUFFER"."MODE SELECTION" = 1) AND ((("BUFFER".PROCESS = 60) AND "AlwaysFALSE") OR (("BUFFER".PROCESS = 190) AND "AlwaysFALSE") OR (("BUFFER".PROCESS = 370) AND "AlwaysFALSE") OR (("BUFFER".PROCESS = 470) AND "AlwaysFALSE") OR (("BUFFER".PROCESS = 590) AND "AlwaysFALSE") OR ("BUFFER".PROCESS = 750) OR ("BUFFER".PROCESS = 850)))) AND NOT "CYCLE PAUSE" AND NOT "ERROR";
END_REGION

REGION Network 18: "PNEUMATIC_VALVE-14" (PBFV-14)
   RUNG wire#powerrail
      Contact( "AlwaysTRUE" )
      wire#w1
      { S7_Templates := "SrcType := Int" } EQ_Contact(in1 := "BUFFER"."MODE SELECTION", in2 := 2)
      Contact( "MANUAL BIT"."PNV-14" )
      wire#w2
      I_Contact( "CYCLE PAUSE" )
      I_Contact( "ERROR" )
      Coil( "OP"."PNV-14" )
   END_RUNG
   RUNG wire#w1
      { S7_Templates := "SrcType := Int" } EQ_Contact(in1 := "BUFFER"."MODE SELECTION", in2 := 1)
      { S7_Templates := "SrcType := Int" } EQ_Contact(in1 := "BUFFER".PROCESS, in2 := 120)
      Contact( "ACID_BIT" )
   END_RUNG wire#w2
   // the same network as SCL:
   "OP"."PNV-14" := "AlwaysTRUE" AND ((("BUFFER"."MODE SELECTION" = 2) AND "MANUAL BIT"."PNV-14") OR (("BUFFER"."MODE SELECTION" = 1) AND ("BUFFER".PROCESS = 120) AND "ACID_BIT")) AND NOT "CYCLE PAUSE" AND NOT "ERROR";
END_REGION

REGION Network 19: "PNEUMATIC_VALVE-15" (PBFV-15)
   RUNG wire#powerrail
      Contact( "AlwaysTRUE" )
      wire#w1
      { S7_Templates := "SrcType := Int" } EQ_Contact(in1 := "BUFFER"."MODE SELECTION", in2 := 2)
      Contact( "MANUAL BIT"."PNV-15" )
      wire#w2
      I_Contact( "CYCLE PAUSE" )
      I_Contact( "ERROR" )
      Coil( "OP"."PNV-15" )
   END_RUNG
   RUNG wire#w1
      { S7_Templates := "SrcType := Int" } EQ_Contact(in1 := "BUFFER"."MODE SELECTION", in2 := 1)
      { S7_Templates := "SrcType := Int" } EQ_Contact(in1 := "BUFFER".PROCESS, in2 := 120)
      Contact( "ALKALI_BIT" )
   END_RUNG wire#w2
   // the same network as SCL:
   "OP"."PNV-15" := "AlwaysTRUE" AND ((("BUFFER"."MODE SELECTION" = 2) AND "MANUAL BIT"."PNV-15") OR (("BUFFER"."MODE SELECTION" = 1) AND ("BUFFER".PROCESS = 120) AND "ALKALI_BIT")) AND NOT "CYCLE PAUSE" AND NOT "ERROR";
END_REGION

REGION Network 20: "PNEUMATIC_VALVE-16" (PBFV-16)
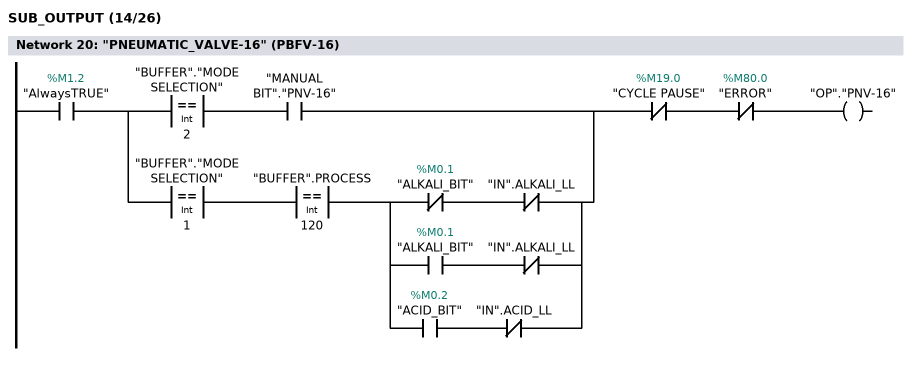
   RUNG wire#powerrail
      Contact( "AlwaysTRUE" )
      wire#w1
      { S7_Templates := "SrcType := Int" } EQ_Contact(in1 := "BUFFER"."MODE SELECTION", in2 := 2)
      Contact( "MANUAL BIT"."PNV-16" )
      wire#w2
      I_Contact( "CYCLE PAUSE" )
      I_Contact( "ERROR" )
      Coil( "OP"."PNV-16" )
   END_RUNG
   RUNG wire#w1
      { S7_Templates := "SrcType := Int" } EQ_Contact(in1 := "BUFFER"."MODE SELECTION", in2 := 1)
      { S7_Templates := "SrcType := Int" } EQ_Contact(in1 := "BUFFER".PROCESS, in2 := 120)
      wire#w3
      I_Contact( "ALKALI_BIT" )
      I_Contact( "IN".ALKALI_LL )
   END_RUNG wire#w2
   RUNG wire#w3
      Contact( "ALKALI_BIT" )
      I_Contact( "IN".ALKALI_LL )
   END_RUNG wire#w2
   RUNG wire#w3
      Contact( "ACID_BIT" )
      I_Contact( "IN".ACID_LL )
   END_RUNG wire#w2
   // the same network as SCL:
   "OP"."PNV-16" := "AlwaysTRUE" AND ((("BUFFER"."MODE SELECTION" = 2) AND "MANUAL BIT"."PNV-16") OR (("BUFFER"."MODE SELECTION" = 1) AND ("BUFFER".PROCESS = 120) AND ((NOT "ALKALI_BIT" AND NOT "IN".ALKALI_LL) OR ("ALKALI_BIT" AND NOT "IN".ALKALI_LL) OR ("ACID_BIT" AND NOT "IN".ACID_LL)))) AND NOT "CYCLE PAUSE" AND NOT "ERROR";
END_REGION

REGION Network 21: "PNEUMATIC_VALVE-17" (PBFV-17) MFG1- MIXING
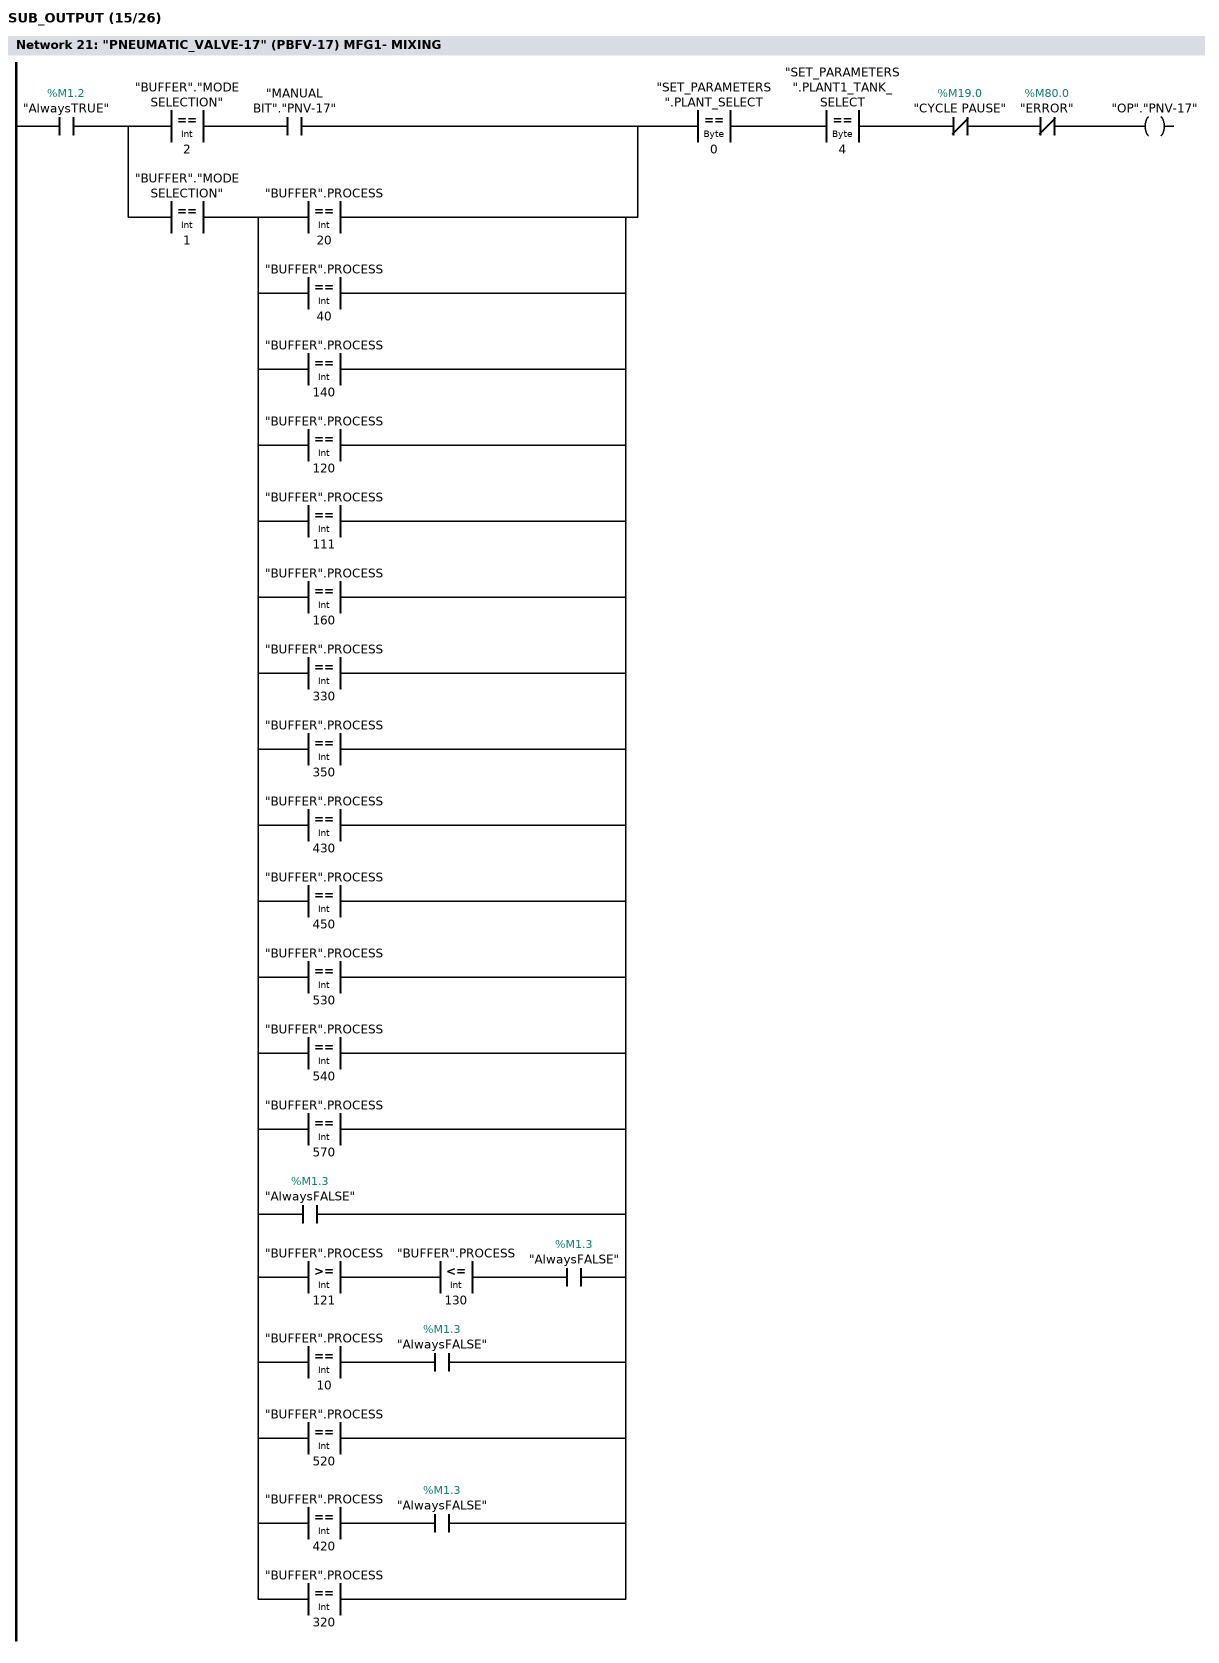
   RUNG wire#powerrail
      Contact( "AlwaysTRUE" )
      wire#w1
      { S7_Templates := "SrcType := Int" } EQ_Contact(in1 := "BUFFER"."MODE SELECTION", in2 := 2)
      Contact( "MANUAL BIT"."PNV-17" )
      wire#w2
      { S7_Templates := "SrcType := Byte" } EQ_Contact(in1 := "SET_PARAMETERS".PLANT_SELECT, in2 := 0)
      { S7_Templates := "SrcType := Byte" } EQ_Contact(in1 := "SET_PARAMETERS".PLANT1_TANK_SELECT, in2 := 4)
      I_Contact( "CYCLE PAUSE" )
      I_Contact( "ERROR" )
      Coil( "OP"."PNV-17" )
   END_RUNG
   RUNG wire#w1
      { S7_Templates := "SrcType := Int" } EQ_Contact(in1 := "BUFFER"."MODE SELECTION", in2 := 1)
      wire#w3
      { S7_Templates := "SrcType := Int" } EQ_Contact(in1 := "BUFFER".PROCESS, in2 := 20)
   END_RUNG wire#w2
   RUNG wire#w3
      { S7_Templates := "SrcType := Int" } EQ_Contact(in1 := "BUFFER".PROCESS, in2 := 40)
   END_RUNG wire#w2
   RUNG wire#w3
      { S7_Templates := "SrcType := Int" } EQ_Contact(in1 := "BUFFER".PROCESS, in2 := 140)
   END_RUNG wire#w2
   RUNG wire#w3
      { S7_Templates := "SrcType := Int" } EQ_Contact(in1 := "BUFFER".PROCESS, in2 := 120)
   END_RUNG wire#w2
   RUNG wire#w3
      { S7_Templates := "SrcType := Int" } EQ_Contact(in1 := "BUFFER".PROCESS, in2 := 111)
   END_RUNG wire#w2
   RUNG wire#w3
      { S7_Templates := "SrcType := Int" } EQ_Contact(in1 := "BUFFER".PROCESS, in2 := 160)
   END_RUNG wire#w2
   RUNG wire#w3
      { S7_Templates := "SrcType := Int" } EQ_Contact(in1 := "BUFFER".PROCESS, in2 := 330)
   END_RUNG wire#w2
   RUNG wire#w3
      { S7_Templates := "SrcType := Int" } EQ_Contact(in1 := "BUFFER".PROCESS, in2 := 350)
   END_RUNG wire#w2
   RUNG wire#w3
      { S7_Templates := "SrcType := Int" } EQ_Contact(in1 := "BUFFER".PROCESS, in2 := 430)
   END_RUNG wire#w2
   RUNG wire#w3
      { S7_Templates := "SrcType := Int" } EQ_Contact(in1 := "BUFFER".PROCESS, in2 := 450)
   END_RUNG wire#w2
   RUNG wire#w3
      { S7_Templates := "SrcType := Int" } EQ_Contact(in1 := "BUFFER".PROCESS, in2 := 530)
   END_RUNG wire#w2
   RUNG wire#w3
      { S7_Templates := "SrcType := Int" } EQ_Contact(in1 := "BUFFER".PROCESS, in2 := 540)
   END_RUNG wire#w2
   RUNG wire#w3
      { S7_Templates := "SrcType := Int" } EQ_Contact(in1 := "BUFFER".PROCESS, in2 := 570)
   END_RUNG wire#w2
   RUNG wire#w3
      Contact( "AlwaysFALSE" )
   END_RUNG wire#w2
   RUNG wire#w3
      { S7_Templates := "SrcType := Int" } GE_Contact(in1 := "BUFFER".PROCESS, in2 := 121)
      { S7_Templates := "SrcType := Int" } LE_Contact(in1 := "BUFFER".PROCESS, in2 := 130)
      Contact( "AlwaysFALSE" )
   END_RUNG wire#w2
   RUNG wire#w3
      { S7_Templates := "SrcType := Int" } EQ_Contact(in1 := "BUFFER".PROCESS, in2 := 10)
      Contact( "AlwaysFALSE" )
   END_RUNG wire#w2
   RUNG wire#w3
      { S7_Templates := "SrcType := Int" } EQ_Contact(in1 := "BUFFER".PROCESS, in2 := 520)
   END_RUNG wire#w2
   RUNG wire#w3
      { S7_Templates := "SrcType := Int" } EQ_Contact(in1 := "BUFFER".PROCESS, in2 := 420)
      Contact( "AlwaysFALSE" )
   END_RUNG wire#w2
   RUNG wire#w3
      { S7_Templates := "SrcType := Int" } EQ_Contact(in1 := "BUFFER".PROCESS, in2 := 320)
   END_RUNG wire#w2
   // the same network as SCL:
   "OP"."PNV-17" := "AlwaysTRUE" AND ((("BUFFER"."MODE SELECTION" = 2) AND "MANUAL BIT"."PNV-17") OR (("BUFFER"."MODE SELECTION" = 1) AND (("BUFFER".PROCESS = 20) OR ("BUFFER".PROCESS = 40) OR ("BUFFER".PROCESS = 140) OR ("BUFFER".PROCESS = 120) OR ("BUFFER".PROCESS = 111) OR ("BUFFER".PROCESS = 160) OR ("BUFFER".PROCESS = 330) OR ("BUFFER".PROCESS = 350) OR ("BUFFER".PROCESS = 430) OR ("BUFFER".PROCESS = 450) OR ("BUFFER".PROCESS = 530) OR ("BUFFER".PROCESS = 540) OR ("BUFFER".PROCESS = 570) OR "AlwaysFALSE" OR (("BUFFER".PROCESS >= 121) AND ("BUFFER".PROCESS <= 130) AND "AlwaysFALSE") OR (("BUFFER".PROCESS = 10) AND "AlwaysFALSE") OR ("BUFFER".PROCESS = 520) OR (("BUFFER".PROCESS = 420) AND "AlwaysFALSE") OR ("BUFFER".PROCESS = 320)))) AND ("SET_PARAMETERS".PLANT_SELECT = 0) AND ("SET_PARAMETERS".PLANT1_TANK_SELECT = 4) AND NOT "CYCLE PAUSE" AND NOT "ERROR";
END_REGION

REGION Network 22: only use manual operated "PNEUMATIC_VALVE-18" (PBFV-18)
